C01810=1180.167,97.495,-51.204,-178.948,6.146,148.795
C01811=1180.172,97.245,-51.186,-178.951,6.145,148.796
C01812=1180.177,96.996,-51.166,-178.954,6.143,148.797
C01813=1180.182,96.747,-51.148,-178.957,6.142,148.797
C01814=1180.187,96.498,-51.130,-178.959,6.141,148.798
C01815=1180.192,96.249,-51.112,-178.962,6.139,148.798
C01816=1180.197,95.999,-51.094,-178.964,6.139,148.799
C01817=1180.201,95.750,-51.076,-178.967,6.137,148.799
C01818=1180.206,95.500,-51.058,-178.970,6.136,148.800
C01819=1180.211,95.251,-51.040,-178.973,6.135,148.800
C01820=1180.217,95.002,-51.021,-178.975,6.134,148.801
C01821=1180.221,94.753,-51.003,-178.978,6.132,148.801
C01822=1180.226,94.503,-50.985,-178.980,6.132,148.802
C01823=1180.231,94.254,-50.967,-178.983,6.130,148.802
C01824=1180.236,94.004,-50.949,-178.985,6.129,148.803
C01825=1180.240,93.755,-50.931,-178.989,6.128,148.803
C01826=1180.245,93.506,-50.913,-178.991,6.127,148.804
C01827=1180.250,93.257,-50.895,-178.993,6.125,148.804
C01828=1180.255,93.008,-50.877,-178.996,6.125,148.805
C01829=1180.260,92.758,-50.859,-178.999,6.123,148.805
C01830=1180.264,92.509,-50.841,-179.002,6.122,148.806
C01831=1180.269,92.259,-50.823,-179.004,6.121,148.806
C01832=1180.274,92.010,-50.805,-179.007,6.119,148.807
C01833=1180.279,91.761,-50.787,-179.009,6.118,148.807
C01834=1180.284,91.512,-50.769,-179.012,6.117,148.808
C01835=1180.289,91.263,-50.751,-179.015,6.116,148.808
C01836=1180.294,91.013,-50.734,-179.017,6.114,148.809
C01837=1180.299,90.764,-50.716,-179.020,6.114,148.809
C01838=1180.304,90.515,-50.698,-179.023,6.112,148.810
C01839=1180.309,90.265,-50.680,-179.025,6.112,148.811
C01840=1180.313,90.016,-50.661,-179.028,6.110,148.811
C01841=1180.318,89.766,-50.643,-179.030,6.109,148.811
C01842=1180.323,89.517,-50.625,-179.034,6.108,148.812
C01843=1180.328,89.267,-50.608,-179.036,6.107,148.812
C01844=1180.333,89.018,-50.590,-179.039,6.105,148.813
C01845=1180.338,88.769,-50.572,-179.041,6.105,148.814
C01846=1180.342,88.520,-50.555,-179.044,6.103,148.814
C01847=1180.347,88.271,-50.537,-179.046,6.102,148.815
C01848=1180.352,88.021,-50.520,-179.050,6.101,148.815
C01849=1180.357,87.772,-50.502,-179.052,6.100,148.816
C01850=1180.362,87.523,-50.484,-179.054,6.099,148.816
C01851=1180.367,87.274,-50.466,-179.057,6.098,148.817
C01852=1180.372,87.024,-50.448,-179.059,6.097,148.817
C01853=1180.377,86.775,-50.430,-179.062,6.096,148.818
C01854=1180.382,86.526,-50.412,-179.064,6.095,148.818
C01855=1180.387,86.276,-50.396,-179.068,6.093,148.819
C01856=1180.392,86.027,-50.378,-179.070,6.092,148.819
C01857=1180.397,85.778,-50.360,-179.073,6.091,148.820
C01858=1180.402,85.528,-50.343,-179.075,6.090,148.820
C01859=1180.407,85.279,-50.325,-179.078,6.089,148.821
C01860=1180.412,85.030,-50.307,-179.081,6.088,148.821
C01861=1180.416,84.780,-50.290,-179.083,6.086,148.822
C01862=1180.421,84.531,-50.272,-179.086,6.086,148.823
C01863=1180.426,84.282,-50.254,-179.089,6.084,148.823
C01864=1180.431,84.032,-50.237,-179.091,6.083,148.824
C01865=1180.436,83.783,-50.219,-179.094,6.082,148.824
C01866=1180.440,83.533,-50.202,-179.097,6.081,148.825
C01867=1180.445,83.284,-50.184,-179.099,6.080,148.825
C01868=1180.450,83.035,-50.166,-179.102,6.079,148.826
C01869=1180.456,82.785,-50.149,-179.104,6.078,148.826
C01870=1180.460,82.536,-50.131,-179.107,6.077,148.827
C01871=1180.465,82.286,-50.114,-179.109,6.076,148.827
C01872=1180.470,82.037,-50.096,-179.113,6.074,148.828
C01873=1180.475,81.787,-50.079,-179.115,6.073,148.828
C01874=1180.479,81.539,-50.062,-179.118,6.072,148.829
C01875=1180.484,81.289,-50.044,-179.120,6.071,148.829
C01876=1180.489,81.040,-50.026,-179.123,6.071,148.830
C01877=1180.495,80.771,-50.008,-179.125,6.069,148.830
C01878=1180.500,80.504,-49.989,-179.129,6.068,148.831
C01879=1180.505,80.235,-49.970,-179.131,6.067,148.832
C01880=1180.511,79.966,-49.952,-179.134,6.065,148.832
C01881=1180.516,79.717,-49.934,-179.137,6.065,148.833
C01882=1180.520,79.468,-49.918,-179.139,6.063,148.833
C01883=1180.525,79.219,-49.900,-179.142,6.063,148.834
C01884=1180.531,78.969,-49.882,-179.145,6.061,148.834
C01885=1180.535,78.719,-49.866,-179.147,6.060,148.835
C01886=1180.540,78.470,-49.848,-179.150,6.059,148.835
C01887=1180.545,78.220,-49.830,-179.153,6.058,148.836
C01888=1180.550,77.972,-49.813,-179.155,6.057,148.837
C01889=1180.555,77.722,-49.796,-179.158,6.056,148.837
C01890=1180.560,77.473,-49.779,-179.160,6.055,148.838
C01891=1180.565,77.224,-49.761,-179.163,6.054,148.838
C01892=1180.570,76.974,-49.744,-179.166,6.053,148.839
C01893=1180.574,76.724,-49.727,-179.168,6.052,148.839
C01894=1180.579,76.475,-49.710,-179.171,6.050,148.840
C01895=1180.584,76.227,-49.693,-179.174,6.050,148.840
C01896=1180.589,75.977,-49.676,-179.176,6.048,148.841
C01897=1180.594,75.728,-49.658,-179.179,6.048,148.841
C01898=1180.599,75.478,-49.641,-179.182,6.046,148.842
C01899=1180.604,75.228,-49.624,-179.184,6.045,148.843
C01900=1180.609,74.979,-49.607,-179.186,6.045,148.843
C01901=1180.614,74.730,-49.590,-179.190,6.043,148.844
C01902=1180.619,74.481,-49.573,-179.192,6.042,148.844
C01903=1180.624,74.231,-49.556,-179.195,6.041,148.845
C01904=1180.628,73.982,-49.539,-179.197,6.040,148.845
C01905=1180.633,73.732,-49.521,-179.200,6.040,148.846
C01906=1180.639,73.483,-49.504,-179.202,6.038,148.846
C01907=1180.643,73.234,-49.488,-179.205,6.037,148.847
C01908=1180.649,72.984,-49.470,-179.207,6.036,148.847
C01909=1180.653,72.735,-49.454,-179.210,6.035,148.848
C01910=1180.658,72.485,-49.436,-179.213,6.034,148.848
C01911=1180.663,72.237,-49.419,-179.216,6.033,148.849
C01912=1180.668,71.987,-49.403,-179.218,6.032,148.850
C01913=1180.673,71.737,-49.385,-179.221,6.031,148.850
C01914=1180.677,71.488,-49.369,-179.223,6.030,148.851
C01915=1180.683,71.239,-49.352,-179.226,6.029,148.851
C01916=1180.688,70.989,-49.335,-179.229,6.027,148.852
C01917=1180.693,70.739,-49.318,-179.231,6.027,148.852
C01918=1180.697,70.491,-49.301,-179.233,6.026,148.853
C01919=1180.703,70.241,-49.284,-179.237,6.025,148.853
C01920=1180.707,69.992,-49.267,-179.239,6.024,148.854
C01921=1180.712,69.743,-49.250,-179.241,6.023,148.855
C01922=1180.718,69.493,-49.233,-179.244,6.022,148.855
C01923=1180.722,69.244,-49.217,-179.247,6.021,148.856
C01924=1180.727,68.994,-49.199,-179.250,6.020,148.856
C01925=1180.732,68.745,-49.183,-179.252,6.019,148.857
C01926=1180.737,68.496,-49.167,-179.255,6.018,148.857
C01927=1180.742,68.246,-49.149,-179.257,6.017,148.858
C01928=1180.747,67.997,-49.133,-179.260,6.016,148.858
C01929=1180.752,67.748,-49.116,-179.262,6.015,148.859
C01930=1180.757,67.498,-49.099,-179.265,6.014,148.860
C01931=1180.761,67.249,-49.082,-179.268,6.013,148.860
C01932=1180.767,66.999,-49.065,-179.270,6.012,148.861
C01933=1180.772,66.750,-49.049,-179.273,6.011,148.861
C01934=1180.776,66.500,-49.032,-179.276,6.010,148.862
C01935=1180.781,66.251,-49.015,-179.278,6.009,148.862
C01936=1180.786,66.002,-48.999,-179.281,6.008,148.863
C01937=1180.791,65.752,-48.982,-179.283,6.007,148.863
C01938=1180.796,65.503,-48.965,-179.286,6.007,148.864
C01939=1180.802,65.253,-48.949,-179.289,6.005,148.865
C01940=1180.806,65.004,-48.932,-179.291,6.004,148.865
C01941=1180.810,64.754,-48.916,-179.294,6.003,148.866
C01942=1180.816,64.505,-48.899,-179.296,6.002,148.866
C01943=1180.821,64.256,-48.882,-179.299,6.002,148.867
C01944=1180.826,64.007,-48.866,-179.302,6.000,148.867
C01945=1180.830,63.757,-48.849,-179.304,5.999,148.868
C01946=1180.836,63.507,-48.833,-179.307,5.998,148.868
C01947=1180.841,63.258,-48.816,-179.310,5.997,148.869
C01948=1180.845,63.009,-48.800,-179.312,5.997,148.870
C01949=1180.850,62.759,-48.783,-179.315,5.996,148.870
C01950=1180.856,62.510,-48.766,-179.318,5.994,148.871
C01951=1180.860,62.261,-48.749,-179.320,5.993,148.871
C01952=1180.866,62.011,-48.734,-179.323,5.993,148.872
C01953=1180.870,61.762,-48.717,-179.325,5.992,148.872
C01954=1180.875,61.512,-48.700,-179.328,5.991,148.873
C01955=1180.880,61.263,-48.684,-179.330,5.990,148.873
C01956=1180.885,61.013,-48.668,-179.333,5.989,148.874
C01957=1180.890,60.764,-48.651,-179.336,5.988,148.875
C01958=1180.895,60.515,-48.635,-179.338,5.987,148.875
C01959=1180.900,60.266,-48.618,-179.341,5.987,148.876
C01960=1180.905,60.016,-48.602,-179.343,5.985,148.876
C01961=1180.910,59.766,-48.585,-179.346,5.984,148.877
C01962=1180.915,59.517,-48.569,-179.348,5.984,148.877
C01963=1180.920,59.267,-48.553,-179.351,5.982,148.878
C01964=1180.925,59.018,-48.537,-179.354,5.981,148.878
C01965=1180.929,58.769,-48.520,-179.356,5.981,148.879
C01966=1180.935,58.520,-48.504,-179.359,5.979,148.880
C01967=1180.940,58.270,-48.487,-179.362,5.979,148.880
C01968=1180.945,58.021,-48.471,-179.364,5.978,148.881
C01969=1180.950,57.771,-48.455,-179.366,5.977,148.881
C01970=1180.955,57.522,-48.438,-179.370,5.976,148.882
C01971=1180.960,57.272,-48.423,-179.372,5.975,148.882
C01972=1180.965,57.023,-48.406,-179.374,5.974,148.883
C01973=1180.969,56.774,-48.390,-179.378,5.973,148.884
C01974=1180.975,56.524,-48.374,-179.380,5.972,148.884
C01975=1180.979,56.275,-48.357,-179.382,5.972,148.885
C01976=1180.984,56.025,-48.342,-179.385,5.971,148.885
C01977=1180.990,55.776,-48.324,-179.388,5.969,148.886
C01978=1180.995,55.526,-48.309,-179.390,5.969,148.886
C01979=1180.999,55.277,-48.292,-179.393,5.968,148.887
C01980=1181.005,55.027,-48.277,-179.396,5.967,148.888
C01981=1181.010,54.759,-48.258,-179.398,5.966,148.888
C01982=1181.015,54.490,-48.241,-179.401,5.965,148.889
C01983=1181.021,54.222,-48.224,-179.404,5.964,148.889
C01984=1181.026,53.953,-48.207,-179.406,5.964,148.890
C01985=1181.031,53.704,-48.191,-179.409,5.962,148.891
C01986=1181.036,53.454,-48.175,-179.412,5.961,148.891
C01987=1181.041,53.205,-48.159,-179.414,5.961,148.892
C01988=1181.046,52.956,-48.143,-179.417,5.960,148.892
C01989=1181.050,52.706,-48.126,-179.420,5.959,148.893
C01990=1181.056,52.457,-48.111,-179.422,5.958,148.893
C01991=1181.060,52.207,-48.094,-179.425,5.957,148.894
C01992=1181.066,51.958,-48.078,-179.427,5.956,148.895
C01993=1181.071,51.708,-48.063,-179.430,5.955,148.895
C01994=1181.076,51.459,-48.046,-179.433,5.954,148.896
C01995=1181.081,51.210,-48.031,-179.435,5.954,148.896
C01996=1181.085,50.960,-48.014,-179.438,5.952,148.897
C01997=1181.091,50.711,-47.998,-179.440,5.951,148.897
C01998=1181.095,50.461,-47.983,-179.443,5.951,148.898
C01999=1181.100,50.212,-47.967,-179.445,5.950,148.899
C02000=1181.105,49.963,-47.951,-179.448,5.949,148.899
C02001=1181.110,49.713,-47.935,-179.451,5.948,148.900
C02002=1181.115,49.464,-47.919,-179.453,5.947,148.900
C02003=1181.120,49.214,-47.903,-179.456,5.947,148.901
C02004=1181.125,48.964,-47.887,-179.459,5.945,148.902
C02005=1181.130,48.716,-47.871,-179.461,5.945,148.902
C02006=1181.135,48.465,-47.855,-179.464,5.944,148.903
C02007=1181.140,48.216,-47.840,-179.466,5.943,148.903
C02008=1181.145,47.967,-47.824,-179.469,5.942,148.904
C02009=1181.150,47.717,-47.808,-179.472,5.941,148.905
C02010=1181.155,47.468,-47.792,-179.474,5.940,148.905
C02011=1181.160,47.219,-47.777,-179.476,5.940,148.906
C02012=1181.165,46.969,-47.761,-179.479,5.939,148.906
C02013=1181.170,46.720,-47.745,-179.482,5.938,148.907
C02014=1181.175,46.471,-47.729,-179.484,5.937,148.907
C02015=1181.180,46.221,-47.713,-179.487,5.936,148.908
C02016=1181.185,45.971,-47.698,-179.489,5.936,148.909
C02017=1181.191,45.722,-47.682,-179.492,5.934,148.909
C02018=1181.194,45.473,-47.666,-179.495,5.934,148.910
C02019=1181.200,45.223,-47.651,-179.497,5.933,148.910
C02020=1181.205,44.974,-47.635,-179.499,5.932,148.911
C02021=1181.210,44.724,-47.619,-179.503,5.931,148.911
C02022=1181.215,44.474,-47.603,-179.505,5.930,148.912
C02023=1181.220,44.225,-47.588,-179.507,5.930,148.913
C02024=1181.225,43.975,-47.572,-179.510,5.929,148.913
C02025=1181.230,43.726,-47.556,-179.512,5.928,148.914
C02026=1181.235,43.477,-47.541,-179.515,5.927,148.914
C02027=1181.239,43.227,-47.525,-179.518,5.926,148.915
C02028=1181.245,42.978,-47.510,-179.520,5.926,148.915
C02029=1181.250,42.728,-47.494,-179.523,5.925,148.916
C02030=1181.255,42.479,-47.478,-179.525,5.924,148.917
C02031=1181.259,42.229,-47.463,-179.528,5.923,148.917
C02032=1181.265,41.980,-47.447,-179.531,5.922,148.918
C02033=1181.270,41.730,-47.432,-179.533,5.921,148.918
C02034=1181.275,41.481,-47.417,-179.536,5.921,148.919
C02035=1181.280,41.231,-47.401,-179.538,5.920,148.920
C02036=1181.285,40.982,-47.385,-179.541,5.919,148.920
C02037=1181.290,40.733,-47.370,-179.544,5.918,148.921
C02038=1181.295,40.483,-47.355,-179.546,5.917,148.921
C02039=1181.300,40.233,-47.339,-179.548,5.917,148.922
C02040=1181.304,39.984,-47.324,-179.551,5.916,148.923
C02041=1181.310,39.735,-47.308,-179.554,5.915,148.923
C02042=1181.315,39.485,-47.293,-179.557,5.914,148.924
C02043=1181.320,39.236,-47.278,-179.559,5.914,148.924
C02044=1181.325,38.986,-47.262,-179.561,5.913,148.925
C02045=1181.330,38.737,-47.246,-179.564,5.912,148.926
C02046=1181.335,38.487,-47.231,-179.567,5.911,148.926
C02047=1181.340,38.238,-47.216,-179.569,5.910,148.927
C02048=1181.346,37.989,-47.200,-179.572,5.910,148.927
C02049=1181.350,37.739,-47.185,-179.574,5.909,148.928
C02050=1181.355,37.489,-47.170,-179.577,5.908,148.928
C02051=1181.360,37.240,-47.155,-179.579,5.908,148.929
C02052=1181.365,36.990,-47.139,-179.582,5.906,148.930
C02053=1181.371,36.741,-47.124,-179.585,5.906,148.930
C02054=1181.375,36.491,-47.108,-179.587,5.905,148.931
C02055=1181.380,36.242,-47.093,-179.590,5.904,148.931
C02056=1181.385,35.993,-47.078,-179.592,5.904,148.932
C02057=1181.390,35.743,-47.063,-179.594,5.903,148.932
C02058=1181.395,35.494,-47.048,-179.598,5.902,148.933
C02059=1181.400,35.244,-47.032,-179.600,5.901,148.934
C02060=1181.405,34.994,-47.017,-179.602,5.900,148.934
C02061=1181.410,34.745,-47.001,-179.605,5.900,148.935
C02062=1181.416,34.495,-46.986,-179.608,5.899,148.936
C02063=1181.420,34.246,-46.971,-179.610,5.898,148.936
C02064=1181.426,33.996,-46.956,-179.613,5.897,148.937
C02065=1181.430,33.747,-46.941,-179.616,5.896,148.937
C02066=1181.436,33.497,-46.926,-179.618,5.896,148.938
C02067=1181.441,33.248,-46.911,-179.621,5.895,148.939
C02068=1181.445,32.998,-46.895,-179.623,5.895,148.939
C02069=1181.450,32.749,-46.880,-179.625,5.894,148.940
C02070=1181.456,32.499,-46.865,-179.629,5.892,148.940
C02071=1181.460,32.250,-46.850,-179.631,5.892,148.941
C02072=1181.465,32.001,-46.835,-179.633,5.891,148.941
C02073=1181.471,31.751,-46.820,-179.636,5.891,148.942
C02074=1181.475,31.502,-46.805,-179.638,5.890,148.943
C02075=1181.481,31.252,-46.790,-179.641,5.889,148.943
C02076=1181.485,31.003,-46.775,-179.643,5.889,148.944
C02077=1181.491,30.753,-46.760,-179.646,5.887,148.944
C02078=1181.495,30.503,-46.744,-179.649,5.887,148.945
C02079=1181.500,30.254,-46.730,-179.652,5.886,148.946
C02080=1181.506,30.004,-46.715,-179.654,5.885,148.946
C02081=1181.510,29.755,-46.700,-179.656,5.885,148.947
C02082=1181.516,29.505,-46.685,-179.659,5.884,148.948
C02083=1181.521,29.256,-46.670,-179.661,5.883,148.948
C02084=1181.526,29.007,-46.654,-179.664,5.882,148.949
C02085=1181.531,28.738,-46.638,-179.667,5.882,148.949
C02086=1181.536,28.469,-46.623,-179.670,5.881,148.950
C02087=1181.542,28.200,-46.606,-179.672,5.880,148.951
C02088=1181.547,27.931,-46.591,-179.675,5.879,148.951
C02089=1181.553,27.682,-46.575,-179.678,5.878,148.952
C02090=1181.557,27.432,-46.561,-179.680,5.878,148.953
C02091=1181.562,27.183,-46.546,-179.682,5.877,148.953
C02092=1181.568,26.933,-46.531,-179.685,5.877,148.954
C02093=1181.572,26.684,-46.516,-179.688,5.876,148.954
C02094=1181.577,26.434,-46.502,-179.690,5.875,148.955
C02095=1181.583,26.185,-46.486,-179.693,5.874,148.955
C02096=1181.588,25.935,-46.472,-179.696,5.873,148.956
C02097=1181.592,25.686,-46.457,-179.698,5.873,148.957
C02098=1181.598,25.436,-46.442,-179.701,5.872,148.957
C02099=1181.603,25.187,-46.427,-179.703,5.872,148.958
C02100=1181.608,24.937,-46.413,-179.705,5.871,148.958
C02101=1181.612,24.688,-46.398,-179.708,5.870,148.959
C02102=1181.618,24.438,-46.383,-179.711,5.870,148.960
C02103=1181.623,24.188,-46.369,-179.713,5.869,148.960
C02104=1181.628,23.939,-46.354,-179.716,5.868,148.961
C02105=1181.633,23.689,-46.339,-179.719,5.867,148.962
C02106=1181.638,23.440,-46.324,-179.721,5.866,148.962
C02107=1181.643,23.190,-46.309,-179.724,5.866,148.963
C02108=1181.648,22.941,-46.295,-179.726,5.865,148.963
C02109=1181.653,22.691,-46.280,-179.728,5.864,148.964
C02110=1181.658,22.442,-46.265,-179.731,5.864,148.965
C02111=1181.663,22.193,-46.250,-179.734,5.863,148.965
C02112=1181.668,21.943,-46.236,-179.736,5.863,148.966
C02113=1181.673,21.694,-46.222,-179.738,5.862,148.966
C02114=1181.679,21.444,-46.207,-179.741,5.862,148.967
C02115=1181.684,21.195,-46.192,-179.743,5.861,148.967
C02116=1181.689,20.945,-46.178,-179.747,5.859,148.968
C02117=1181.693,20.696,-46.163,-179.749,5.859,148.969
C02118=1181.698,20.446,-46.149,-179.751,5.858,148.969
C02119=1181.704,20.196,-46.134,-179.754,5.858,148.970
C02120=1181.709,19.946,-46.120,-179.757,5.857,148.971
C02121=1181.714,19.697,-46.105,-179.759,5.856,148.971
C02122=1181.719,19.448,-46.090,-179.761,5.856,148.972
C02123=1181.724,19.198,-46.076,-179.764,5.855,148.972
C02124=1181.729,18.949,-46.062,-179.766,5.854,148.973
C02125=1181.734,18.700,-46.046,-179.769,5.854,148.974
C02126=1181.739,18.450,-46.032,-179.772,5.853,148.974
C02127=1181.744,18.200,-46.018,-179.774,5.853,148.975
C02128=1181.749,17.950,-46.004,-179.777,5.851,148.975
C02129=1181.754,17.701,-45.989,-179.780,5.851,148.976
C02130=1181.759,17.452,-45.974,-179.782,5.850,148.977
C02131=1181.764,17.202,-45.960,-179.784,5.849,148.977
C02132=1181.769,16.952,-45.946,-179.787,5.849,148.978
C02133=1181.774,16.703,-45.932,-179.789,5.848,148.978
C02134=1181.779,16.453,-45.918,-179.792,5.848,148.979
C02135=1181.785,16.204,-45.902,-179.795,5.847,148.980
C02136=1181.790,15.954,-45.888,-179.797,5.846,148.980
C02137=1181.795,15.705,-45.874,-179.799,5.846,148.981
C02138=1181.800,15.455,-45.859,-179.802,5.845,148.982
C02139=1181.805,15.206,-45.845,-179.805,5.845,148.982
C02140=1181.810,14.956,-45.831,-179.807,5.844,148.983
C02141=1181.815,14.706,-45.817,-179.809,5.843,148.983
C02142=1181.820,14.457,-45.802,-179.812,5.843,148.984
C02143=1181.825,14.208,-45.787,-179.814,5.842,148.985
C02144=1181.830,13.958,-45.773,-179.817,5.842,148.985
C02145=1181.835,13.709,-45.759,-179.820,5.841,148.986
C02146=1181.840,13.459,-45.745,-179.822,5.839,148.986
C02147=1181.845,13.210,-45.731,-179.825,5.839,148.987
C02148=1181.850,12.960,-45.716,-179.828,5.839,148.988
C02149=1181.855,12.710,-45.702,-179.830,5.838,148.988
C02150=1181.861,12.461,-45.688,-179.832,5.837,148.989
C02151=1181.866,12.211,-45.674,-179.835,5.837,148.990
C02152=1181.870,11.962,-45.660,-179.837,5.836,148.990
C02153=1181.875,11.712,-45.645,-179.840,5.835,148.991
C02154=1181.881,11.463,-45.632,-179.843,5.835,148.991
C02155=1181.886,11.213,-45.617,-179.845,5.834,148.992
C02156=1181.891,10.964,-45.603,-179.847,5.834,148.993
C02157=1181.896,10.714,-45.589,-179.850,5.833,148.993
C02158=1181.901,10.464,-45.574,-179.853,5.833,148.994
C02159=1181.906,10.215,-45.561,-179.855,5.832,148.994
C02160=1181.911,9.965,-45.546,-179.858,5.831,148.995
C02161=1181.916,9.716,-45.532,-179.860,5.831,148.996
C02162=1181.921,9.466,-45.518,-179.862,5.830,148.996
C02163=1181.926,9.217,-45.505,-179.865,5.829,148.997
C02164=1181.931,8.967,-45.491,-179.868,5.829,148.998
C02165=1181.936,8.717,-45.477,-179.870,5.828,148.998
C02166=1181.942,8.468,-45.463,-179.872,5.828,148.999
C02167=1181.947,8.219,-45.448,-179.875,5.827,148.999
C02168=1181.952,7.969,-45.434,-179.877,5.826,149.000
C02169=1181.957,7.719,-45.420,-179.880,5.826,149.001
C02170=1181.962,7.470,-45.406,-179.883,5.825,149.001
C02171=1181.967,7.220,-45.392,-179.885,5.825,149.002
C02172=1181.972,6.970,-45.379,-179.887,5.824,149.002
C02173=1181.977,6.721,-45.365,-179.890,5.824,149.003
C02174=1181.982,6.472,-45.350,-179.893,5.823,149.004
C02175=1181.987,6.222,-45.336,-179.895,5.822,149.004
C02176=1181.992,5.972,-45.322,-179.898,5.822,149.005
C02177=1181.998,5.723,-45.309,-179.900,5.821,149.006
C02178=1182.002,5.473,-45.295,-179.902,5.820,149.006
C02179=1182.007,5.223,-45.281,-179.905,5.820,149.007
C02180=1182.013,4.974,-45.267,-179.908,5.819,149.007
C02181=1182.018,4.725,-45.253,-179.910,5.819,149.008
C02182=1182.023,4.474,-45.239,-179.912,5.818,149.009
C02183=1182.028,4.226,-45.226,-179.915,5.818,149.009
C02184=1182.033,3.976,-45.211,-179.918,5.817,149.010
C02185=1182.038,3.726,-45.197,-179.920,5.816,149.010
C02186=1182.044,3.477,-45.184,-179.923,5.816,149.011
C02187=1182.048,3.227,-45.170,-179.925,5.815,149.012
C02188=1182.053,2.978,-45.156,-179.927,5.815,149.012
C02189=1182.059,2.709,-45.141,-179.930,5.814,149.013
C02190=1182.064,2.439,-45.126,-179.933,5.814,149.014
C02191=1182.070,2.170,-45.111,-179.936,5.812,149.014
C02192=1182.075,1.901,-45.096,-179.939,5.812,149.015
C02193=1182.081,1.651,-45.083,-179.941,5.811,149.016
C02194=1182.085,1.402,-45.069,-179.943,5.811,149.016
C02195=1182.091,1.153,-45.056,-179.946,5.810,149.017
C02196=1182.096,0.902,-45.042,-179.949,5.810,149.017
C02197=1182.101,0.653,-45.028,-179.951,5.809,149.018
C02198=1182.106,0.404,-45.014,-179.954,5.808,149.019
C02199=1182.111,0.154,-45.001,-179.956,5.808,149.019
C02200=1182.117,-0.095,-44.987,-179.959,5.807,149.020
C02201=1182.121,-0.345,-44.973,-179.961,5.806,149.020
C02202=1182.126,-0.595,-44.960,-179.964,5.806,149.021
C02203=1182.132,-0.844,-44.946,-179.966,5.806,149.022
C02204=1182.136,-1.094,-44.933,-179.968,5.805,149.022
C02205=1182.142,-1.343,-44.919,-179.971,5.805,149.023
C02206=1182.147,-1.594,-44.905,-179.973,5.805,149.024
C02207=1182.151,-1.843,-44.892,-179.976,5.804,149.024
C02208=1182.157,-2.092,-44.878,-179.978,5.803,149.025
C02209=1182.162,-2.342,-44.864,-179.981,5.803,149.026
C02210=1182.167,-2.591,-44.851,-179.983,5.802,149.026
C02211=1182.172,-2.841,-44.837,-179.986,5.801,149.027
C02212=1182.178,-3.090,-44.823,-179.988,5.801,149.027
C02213=1182.182,-3.340,-44.810,-179.991,5.801,149.028
C02214=1182.188,-3.589,-44.797,-179.993,5.800,149.029
C02215=1182.192,-3.839,-44.784,-179.996,5.799,149.029
C02216=1182.198,-4.088,-44.770,-179.998,5.799,149.030
C02217=1182.203,-4.339,-44.756,179.999,5.798,149.031
C02218=1182.207,-4.588,-44.742,179.997,5.797,149.031
C02219=1182.213,-4.838,-44.729,179.994,5.797,149.032
C02220=1182.218,-5.088,-44.716,179.992,5.796,149.032
C02221=1182.223,-5.337,-44.702,179.989,5.796,149.033
C02222=1182.228,-5.587,-44.689,179.987,5.795,149.034
C02223=1182.233,-5.836,-44.675,179.984,5.795,149.034
C02224=1182.238,-6.086,-44.662,179.981,5.794,149.035
C02225=1182.243,-6.335,-44.649,179.979,5.793,149.035
C02226=1182.249,-6.585,-44.635,179.977,5.794,149.036
C02227=1182.254,-6.834,-44.622,179.975,5.793,149.037
C02228=1182.259,-7.084,-44.608,179.972,5.792,149.037
C02229=1182.264,-7.334,-44.596,179.970,5.792,149.038
C02230=1182.269,-7.584,-44.582,179.967,5.792,149.039
C02231=1182.274,-7.833,-44.569,179.965,5.791,149.039
C02232=1182.280,-8.082,-44.555,179.962,5.790,149.040
C02233=1182.284,-8.332,-44.543,179.960,5.790,149.041
C02234=1182.290,-8.581,-44.529,179.957,5.789,149.041
C02235=1182.294,-8.831,-44.516,179.955,5.788,149.042
C02236=1182.300,-9.081,-44.502,179.952,5.788,149.042
C02237=1182.304,-9.330,-44.489,179.949,5.788,149.043
C02238=1182.310,-9.580,-44.476,179.947,5.787,149.044
C02239=1182.315,-9.830,-44.463,179.945,5.786,149.044
C02240=1182.320,-10.079,-44.449,179.942,5.786,149.045
C02241=1182.325,-10.329,-44.436,179.940,5.786,149.046
C02242=1182.331,-10.579,-44.423,179.938,5.785,149.046
C02243=1182.336,-10.828,-44.410,179.935,5.785,149.047
C02244=1182.341,-11.078,-44.396,179.932,5.784,149.047
C02245=1182.346,-11.327,-44.383,179.930,5.783,149.048
C02246=1182.350,-11.577,-44.370,179.928,5.783,149.049
C02247=1182.356,-11.827,-44.357,179.925,5.783,149.049
C02248=1182.360,-12.076,-44.343,179.922,5.782,149.050
C02249=1182.366,-12.326,-44.330,179.920,5.781,149.050
C02250=1182.371,-12.575,-44.317,179.917,5.781,149.051
C02251=1182.377,-12.825,-44.304,179.915,5.780,149.052
C02252=1182.382,-13.075,-44.291,179.913,5.779,149.052
C02253=1182.386,-13.324,-44.278,179.910,5.780,149.053
C02254=1182.392,-13.574,-44.264,179.908,5.779,149.054
C02255=1182.397,-13.823,-44.252,179.905,5.779,149.054
C02256=1182.402,-14.073,-44.239,179.903,5.778,149.055
C02257=1182.407,-14.323,-44.226,179.900,5.778,149.056
C02258=1182.412,-14.573,-44.213,179.898,5.777,149.056
C02259=1182.418,-14.822,-44.199,179.895,5.776,149.057
C02260=1182.423,-15.071,-44.186,179.893,5.776,149.057
C02261=1182.427,-15.321,-44.173,179.890,5.775,149.058
C02262=1182.433,-15.571,-44.160,179.888,5.775,149.059
C02263=1182.438,-15.820,-44.147,179.886,5.775,149.059
C02264=1182.443,-16.070,-44.134,179.883,5.774,149.060
C02265=1182.449,-16.319,-44.121,179.881,5.774,149.061
C02266=1182.454,-16.569,-44.109,179.878,5.773,149.061
C02267=1182.458,-16.819,-44.096,179.876,5.773,149.062
C02268=1182.464,-17.068,-44.082,179.873,5.772,149.062
C02269=1182.469,-17.318,-44.070,179.870,5.772,149.063
C02270=1182.473,-17.567,-44.056,179.868,5.771,149.064
C02271=1182.479,-17.816,-44.044,179.866,5.770,149.064
C02272=1182.484,-18.066,-44.030,179.864,5.771,149.065
C02273=1182.489,-18.316,-44.017,179.861,5.770,149.065
C02274=1182.494,-18.565,-44.005,179.859,5.770,149.066
C02275=1182.500,-18.815,-43.992,179.856,5.769,149.067
C02276=1182.504,-19.065,-43.979,179.854,5.768,149.067
C02277=1182.510,-19.314,-43.966,179.851,5.768,149.068
C02278=1182.515,-19.564,-43.953,179.849,5.767,149.069
C02279=1182.521,-19.813,-43.940,179.846,5.767,149.069
C02280=1182.525,-20.063,-43.927,179.844,5.767,149.070
C02281=1182.530,-20.313,-43.915,179.842,5.766,149.071
C02282=1182.536,-20.563,-43.903,179.839,5.766,149.071
C02283=1182.541,-20.813,-43.889,179.837,5.765,149.072
C02284=1182.546,-21.062,-43.877,179.834,5.765,149.072
C02285=1182.551,-21.312,-43.864,179.832,5.764,149.073
C02286=1182.556,-21.561,-43.851,179.829,5.764,149.074
C02287=1182.561,-21.811,-43.838,179.827,5.763,149.074
C02288=1182.567,-22.061,-43.825,179.825,5.763,149.075
C02289=1182.572,-22.310,-43.813,179.822,5.763,149.076
C02290=1182.577,-22.559,-43.800,179.820,5.762,149.076
C02291=1182.581,-22.809,-43.787,179.817,5.762,149.077
C02292=1182.586,-23.059,-43.774,179.814,5.761,149.078
C02293=1182.593,-23.329,-43.761,179.812,5.761,149.078
C02294=1182.598,-23.598,-43.748,179.809,5.760,149.079
C02295=1182.604,-23.868,-43.733,179.806,5.760,149.080
C02296=1182.609,-24.138,-43.720,179.804,5.759,149.080
C02297=1182.614,-24.387,-43.707,179.802,5.758,149.081
C02298=1182.619,-24.637,-43.694,179.799,5.758,149.082
C02299=1182.625,-24.887,-43.683,179.797,5.758,149.082
C02300=1182.630,-25.136,-43.669,179.795,5.758,149.083
C02301=1182.635,-25.386,-43.656,179.792,5.757,149.083
C02302=1182.640,-25.636,-43.644,179.789,5.757,149.084
C02303=1182.645,-25.885,-43.631,179.787,5.756,149.085
C02304=1182.651,-26.135,-43.619,179.785,5.755,149.085
C02305=1182.655,-26.385,-43.606,179.782,5.755,149.086
C02306=1182.660,-26.634,-43.594,179.780,5.755,149.087
C02307=1182.665,-26.883,-43.581,179.778,5.754,149.087
C02308=1182.671,-27.133,-43.569,179.775,5.754,149.088
C02309=1182.676,-27.383,-43.557,179.772,5.754,149.088
C02310=1182.681,-27.632,-43.544,179.770,5.753,149.089
C02311=1182.686,-27.882,-43.530,179.767,5.752,149.090
C02312=1182.692,-28.132,-43.519,179.765,5.753,149.090
C02313=1182.697,-28.382,-43.506,179.763,5.752,149.091
C02314=1182.702,-28.631,-43.493,179.761,5.751,149.092
C02315=1182.707,-28.881,-43.482,179.758,5.751,149.092
C02316=1182.712,-29.131,-43.469,179.755,5.750,149.093
C02317=1182.717,-29.380,-43.456,179.753,5.750,149.094
C02318=1182.723,-29.630,-43.444,179.751,5.750,149.094
C02319=1182.728,-29.879,-43.431,179.748,5.749,149.095
C02320=1182.733,-30.129,-43.419,179.746,5.749,149.095
C02321=1182.738,-30.379,-43.407,179.744,5.748,149.096
C02322=1182.743,-30.628,-43.394,179.741,5.748,149.097
C02323=1182.748,-30.878,-43.381,179.738,5.747,149.097
C02324=1182.753,-31.128,-43.370,179.736,5.748,149.098
C02325=1182.758,-31.377,-43.357,179.734,5.747,149.099
C02326=1182.764,-31.627,-43.344,179.731,5.746,149.099
C02327=1182.769,-31.877,-43.332,179.729,5.746,149.100
C02328=1182.774,-32.126,-43.320,179.726,5.745,149.100
C02329=1182.780,-32.376,-43.308,179.724,5.745,149.101
C02330=1182.785,-32.625,-43.295,179.722,5.745,149.102
C02331=1182.790,-32.875,-43.283,179.719,5.745,149.102
C02332=1182.795,-33.125,-43.270,179.717,5.744,149.103
C02333=1182.800,-33.374,-43.258,179.714,5.743,149.104
C02334=1182.805,-33.624,-43.246,179.712,5.743,149.104
C02335=1182.810,-33.873,-43.234,179.710,5.743,149.105
C02336=1182.815,-34.123,-43.222,179.707,5.742,149.106
C02337=1182.820,-34.373,-43.210,179.705,5.742,149.106
C02338=1182.826,-34.623,-43.198,179.702,5.741,149.107
C02339=1182.831,-34.872,-43.185,179.700,5.741,149.107
C02340=1182.836,-35.122,-43.173,179.698,5.741,149.108
C02341=1182.841,-35.371,-43.161,179.695,5.741,149.109
C02342=1182.847,-35.621,-43.149,179.693,5.740,149.109
C02343=1182.852,-35.870,-43.136,179.690,5.739,149.110
C02344=1182.857,-36.120,-43.124,179.688,5.739,149.111
C02345=1182.862,-36.370,-43.112,179.686,5.739,149.111
C02346=1182.867,-36.619,-43.100,179.683,5.738,149.112
C02347=1182.872,-36.870,-43.088,179.681,5.738,149.113
C02348=1182.877,-37.119,-43.075,179.678,5.738,149.113
C02349=1182.882,-37.369,-43.064,179.676,5.737,149.114
C02350=1182.887,-37.618,-43.051,179.674,5.737,149.114
C02351=1182.893,-37.868,-43.039,179.671,5.737,149.115
C02352=1182.898,-38.118,-43.026,179.669,5.736,149.116
C02353=1182.903,-38.367,-43.015,179.666,5.735,149.116
C02354=1182.908,-38.617,-43.003,179.664,5.735,149.117
C02355=1182.913,-38.867,-42.991,179.662,5.735,149.117
C02356=1182.919,-39.117,-42.979,179.659,5.734,149.118
C02357=1182.924,-39.366,-42.966,179.657,5.734,149.119
C02358=1182.929,-39.616,-42.954,179.654,5.734,149.120
C02359=1182.934,-39.865,-42.943,179.652,5.734,149.120
C02360=1182.939,-40.115,-42.930,179.650,5.733,149.121
C02361=1182.945,-40.365,-42.919,179.647,5.733,149.121
C02362=1182.950,-40.615,-42.907,179.645,5.732,149.122
C02363=1182.955,-40.864,-42.894,179.642,5.731,149.123
C02364=1182.960,-41.114,-42.883,179.640,5.732,149.123
C02365=1182.965,-41.363,-42.871,179.637,5.731,149.124
C02366=1182.970,-41.613,-42.858,179.635,5.731,149.124
C02367=1182.976,-41.863,-42.846,179.633,5.730,149.125
C02368=1182.980,-42.112,-42.835,179.631,5.730,149.126
C02369=1182.986,-42.362,-42.823,179.628,5.730,149.126
C02370=1182.991,-42.612,-42.811,179.626,5.729,149.127
C02371=1182.997,-42.861,-42.799,179.623,5.729,149.128
C02372=1183.002,-43.110,-42.788,179.621,5.728,149.128
C02373=1183.007,-43.360,-42.776,179.619,5.728,149.129
C02374=1183.012,-43.610,-42.763,179.616,5.728,149.130
C02375=1183.018,-43.860,-42.751,179.613,5.727,149.130
C02376=1183.022,-44.109,-42.740,179.611,5.727,149.131
C02377=1183.028,-44.359,-42.728,179.609,5.727,149.131
C02378=1183.033,-44.609,-42.716,179.606,5.727,149.132
C02379=1183.038,-44.858,-42.704,179.604,5.726,149.133
C02380=1183.043,-45.108,-42.692,179.602,5.725,149.133
C02381=1183.048,-45.358,-42.681,179.600,5.726,149.134
C02382=1183.053,-45.608,-42.669,179.597,5.725,149.135
C02383=1183.058,-45.857,-42.657,179.595,5.724,149.135
C02384=1183.064,-46.107,-42.645,179.592,5.724,149.136
C02385=1183.069,-46.356,-42.634,179.590,5.724,149.137
C02386=1183.074,-46.606,-42.622,179.588,5.724,149.137
C02387=1183.080,-46.856,-42.610,179.585,5.723,149.138
C02388=1183.085,-47.105,-42.599,179.582,5.723,149.139
C02389=1183.090,-47.355,-42.587,179.581,5.723,149.139
C02390=1183.095,-47.605,-42.574,179.578,5.722,149.140
C02391=1183.100,-47.854,-42.563,179.576,5.722,149.140
C02392=1183.105,-48.104,-42.551,179.573,5.721,149.141
C02393=1183.111,-48.354,-42.539,179.571,5.721,149.142
C02394=1183.116,-48.603,-42.528,179.569,5.721,149.142
C02395=1183.121,-48.853,-42.516,179.566,5.720,149.143
C02396=1183.126,-49.103,-42.505,179.564,5.720,149.143
C02397=1183.132,-49.373,-42.492,179.561,5.719,149.144
C02398=1183.138,-49.644,-42.480,179.559,5.720,149.145
C02399=1183.143,-49.914,-42.467,179.556,5.719,149.146
C02400=1183.148,-50.184,-42.454,179.554,5.719,149.146
C02401=1183.154,-50.434,-42.443,179.551,5.718,149.147
C02402=1183.160,-50.683,-42.431,179.549,5.717,149.147
C02403=1183.164,-50.933,-42.420,179.547,5.718,149.148
C02404=1183.170,-51.183,-42.408,179.544,5.717,149.149
C02405=1183.175,-51.432,-42.397,179.542,5.717,149.149
C02406=1183.180,-51.682,-42.385,179.539,5.716,149.150
C02407=1183.185,-51.932,-42.373,179.537,5.717,149.151
C02408=1183.191,-52.181,-42.362,179.535,5.716,149.151
C02409=1183.195,-52.431,-42.351,179.532,5.715,149.152
C02410=1183.201,-52.681,-42.339,179.530,5.715,149.153
C02411=1183.206,-52.931,-42.327,179.528,5.715,149.153
C02412=1183.211,-53.180,-42.315,179.525,5.714,149.154
C02413=1183.217,-53.429,-42.304,179.523,5.714,149.155
C02414=1183.222,-53.679,-42.293,179.521,5.714,149.155
C02415=1183.227,-53.929,-42.281,179.518,5.714,149.156
C02416=1183.232,-54.179,-42.270,179.516,5.713,149.156
C02417=1183.237,-54.429,-42.258,179.513,5.713,149.157
C02418=1183.242,-54.679,-42.247,179.512,5.713,149.158
C02419=1183.247,-54.928,-42.236,179.509,5.712,149.158
C02420=1183.253,-55.178,-42.224,179.506,5.712,149.159
C02421=1183.258,-55.427,-42.213,179.505,5.712,149.159
C02422=1183.263,-55.677,-42.201,179.502,5.711,149.160
C02423=1183.268,-55.926,-42.190,179.499,5.711,149.161
C02424=1183.274,-56.176,-42.178,179.497,5.710,149.161
C02425=1183.278,-56.426,-42.167,179.495,5.711,149.162
C02426=1183.284,-56.676,-42.156,179.492,5.710,149.163
C02427=1183.289,-56.926,-42.145,179.490,5.709,149.163
C02428=1183.295,-57.175,-42.133,179.488,5.710,149.164
C02429=1183.300,-57.425,-42.122,179.485,5.709,149.165
C02430=1183.304,-57.674,-42.110,179.483,5.708,149.165
C02431=1183.310,-57.924,-42.099,179.481,5.708,149.166
C02432=1183.315,-58.174,-42.088,179.479,5.708,149.167
C02433=1183.321,-58.424,-42.076,179.476,5.708,149.167
C02434=1183.325,-58.673,-42.065,179.474,5.707,149.168
C02435=1183.330,-58.923,-42.054,179.472,5.708,149.168
C02436=1183.336,-59.172,-42.042,179.469,5.707,149.169
C02437=1183.341,-59.423,-42.032,179.467,5.706,149.170
C02438=1183.347,-59.672,-42.020,179.465,5.707,149.170
C02439=1183.352,-59.921,-42.009,179.462,5.706,149.171
C02440=1183.357,-60.171,-41.998,179.460,5.705,149.171
C02441=1183.362,-60.422,-41.986,179.457,5.705,149.172
C02442=1183.367,-60.671,-41.975,179.455,5.705,149.173
C02443=1183.372,-60.920,-41.964,179.453,5.705,149.173
C02444=1183.378,-61.170,-41.952,179.450,5.704,149.174
C02445=1183.383,-61.420,-41.942,179.448,5.705,149.175
C02446=1183.388,-61.669,-41.931,179.446,5.704,149.175
C02447=1183.393,-61.919,-41.919,179.443,5.703,149.176
C02448=1183.398,-62.169,-41.908,179.441,5.704,149.177
C02449=1183.404,-62.418,-41.898,179.439,5.703,149.177
C02450=1183.409,-62.668,-41.886,179.436,5.702,149.178
C02451=1183.414,-62.919,-41.875,179.434,5.702,149.179
C02452=1183.419,-63.167,-41.864,179.432,5.702,149.179
C02453=1183.425,-63.417,-41.852,179.429,5.702,149.180
C02454=1183.430,-63.668,-41.842,179.427,5.701,149.180
C02455=1183.435,-63.917,-41.831,179.425,5.701,149.181
C02456=1183.440,-64.166,-41.819,179.422,5.701,149.182
C02457=1183.446,-64.417,-41.808,179.420,5.700,149.182
C02458=1183.451,-64.666,-41.797,179.418,5.700,149.183
C02459=1183.456,-64.915,-41.786,179.416,5.700,149.184
C02460=1183.461,-65.166,-41.775,179.413,5.699,149.184
C02461=1183.467,-65.415,-41.764,179.411,5.699,149.185
C02462=1183.472,-65.665,-41.753,179.409,5.699,149.185
C02463=1183.476,-65.915,-41.742,179.406,5.699,149.186
C02464=1183.482,-66.164,-41.731,179.404,5.699,149.187
C02465=1183.487,-66.414,-41.720,179.402,5.698,149.187
C02466=1183.493,-66.663,-41.709,179.399,5.698,149.188
C02467=1183.498,-66.913,-41.699,179.397,5.698,149.188
C02468=1183.503,-67.163,-41.687,179.395,5.697,149.189
C02469=1183.509,-67.413,-41.676,179.392,5.697,149.190
C02470=1183.513,-67.662,-41.665,179.390,5.697,149.190
C02471=1183.519,-67.912,-41.655,179.388,5.697,149.191
C02472=1183.524,-68.162,-41.644,179.385,5.696,149.192
C02473=1183.529,-68.412,-41.632,179.384,5.696,149.192
C02474=1183.535,-68.661,-41.622,179.381,5.696,149.193
C02475=1183.539,-68.911,-41.610,179.378,5.695,149.194
C02476=1183.545,-69.160,-41.600,179.377,5.695,149.194
C02477=1183.550,-69.410,-41.589,179.374,5.695,149.195
C02478=1183.555,-69.660,-41.578,179.371,5.694,149.196
C02479=1183.561,-69.910,-41.567,179.370,5.694,149.196
C02480=1183.566,-70.160,-41.556,179.367,5.694,149.197
C02481=1183.571,-70.409,-41.546,179.364,5.694,149.197
C02482=1183.576,-70.659,-41.535,179.363,5.694,149.198
C02483=1183.582,-70.908,-41.524,179.360,5.693,149.199
C02484=1183.587,-71.158,-41.512,179.357,5.693,149.199
C02485=1183.592,-71.408,-41.502,179.356,5.693,149.200
C02486=1183.597,-71.657,-41.491,179.353,5.692,149.201
C02487=1183.602,-71.908,-41.480,179.350,5.692,149.201
C02488=1183.608,-72.157,-41.470,179.349,5.692,149.202
C02489=1183.613,-72.407,-41.459,179.346,5.691,149.202
C02490=1183.618,-72.656,-41.449,179.344,5.691,149.203
C02491=1183.624,-72.906,-41.437,179.342,5.691,149.204
C02492=1183.629,-73.156,-41.427,179.339,5.691,149.204
C02493=1183.634,-73.406,-41.416,179.338,5.691,149.205
C02494=1183.639,-73.655,-41.405,179.335,5.690,149.206
C02495=1183.644,-73.905,-41.395,179.332,5.690,149.206
C02496=1183.650,-74.155,-41.384,179.331,5.690,149.207
C02497=1183.655,-74.404,-41.373,179.328,5.689,149.207
C02498=1183.660,-74.654,-41.363,179.325,5.689,149.208
C02499=1183.665,-74.904,-41.352,179.324,5.689,149.209
C02500=1183.671,-75.153,-41.341,179.321,5.689,149.209
C02501=1183.677,-75.425,-41.330,179.318,5.688,149.210
C02502=1183.682,-75.696,-41.318,179.316,5.688,149.211
C02503=1183.688,-75.966,-41.307,179.314,5.688,149.211
C02504=1183.694,-76.237,-41.295,179.311,5.687,149.212
C02505=1183.699,-76.487,-41.285,179.309,5.687,149.213
C02506=1183.704,-76.737,-41.274,179.307,5.687,149.213
C02507=1183.710,-76.987,-41.264,179.305,5.687,149.214
C02508=1183.714,-77.236,-41.252,179.302,5.686,149.215
C02509=1183.720,-77.486,-41.242,179.300,5.687,149.215
C02510=1183.725,-77.736,-41.232,179.298,5.686,149.216
C02511=1183.731,-77.986,-41.221,179.296,5.686,149.216
C02512=1183.735,-78.235,-41.210,179.293,5.685,149.217
C02513=1183.741,-78.485,-41.200,179.291,5.685,149.218
C02514=1183.746,-78.735,-41.189,179.289,5.685,149.218
C02515=1183.752,-78.984,-41.179,179.286,5.684,149.219
C02516=1183.756,-79.234,-41.168,179.284,5.684,149.220
C02517=1183.762,-79.484,-41.158,179.282,5.684,149.220
C02518=1183.767,-79.733,-41.147,179.279,5.684,149.221
C02519=1183.772,-79.983,-41.137,179.277,5.684,149.221
C02520=1183.778,-80.233,-41.127,179.275,5.684,149.222
C02521=1183.783,-80.483,-41.115,179.273,5.683,149.223
C02522=1183.788,-80.732,-41.105,179.270,5.683,149.223
C02523=1183.793,-80.982,-41.095,179.268,5.682,149.224
C02524=1183.799,-81.232,-41.084,179.266,5.682,149.225
C02525=1183.805,-81.481,-41.074,179.263,5.682,149.225
C02526=1183.810,-81.732,-41.064,179.261,5.682,149.226
C02527=1183.815,-81.981,-41.053,179.259,5.682,149.226
C02528=1183.820,-82.231,-41.042,179.257,5.682,149.227
C02529=1183.825,-82.480,-41.032,179.254,5.681,149.228
C02530=1183.830,-82.730,-41.022,179.252,5.681,149.228
C02531=1183.835,-82.980,-41.012,179.250,5.680,149.229
C02532=1183.841,-83.229,-41.002,179.248,5.681,149.230
C02533=1183.846,-83.480,-40.991,179.245,5.680,149.230
C02534=1183.851,-83.729,-40.981,179.243,5.680,149.231
C02535=1183.857,-83.979,-40.971,179.241,5.680,149.231
C02536=1183.862,-84.229,-40.960,179.238,5.680,149.232
C02537=1183.868,-84.479,-40.950,179.236,5.679,149.233
C02538=1183.873,-84.729,-40.939,179.234,5.679,149.233
C02539=1183.877,-84.977,-40.929,179.232,5.678,149.234
C02540=1183.883,-85.227,-40.919,179.230,5.679,149.235
C02541=1183.888,-85.477,-40.908,179.227,5.678,149.235
C02542=1183.893,-85.727,-40.898,179.225,5.678,149.236
C02543=1183.899,-85.976,-40.888,179.223,5.678,149.236
C02544=1183.904,-86.227,-40.877,179.221,5.677,149.237
C02545=1183.909,-86.476,-40.867,179.219,5.678,149.238
C02546=1183.914,-86.726,-40.857,179.216,5.677,149.238
C02547=1183.919,-86.976,-40.847,179.214,5.676,149.239
C02548=1183.925,-87.225,-40.836,179.212,5.677,149.240
C02549=1183.930,-87.475,-40.826,179.209,5.676,149.240
C02550=1183.936,-87.725,-40.816,179.207,5.676,149.241
C02551=1183.940,-87.974,-40.806,179.205,5.676,149.241
C02552=1183.945,-88.224,-40.795,179.203,5.676,149.242
C02553=1183.951,-88.474,-40.785,179.200,5.676,149.243
C02554=1183.957,-88.724,-40.776,179.198,5.675,149.243
C02555=1183.962,-88.974,-40.765,179.196,5.675,149.244
C02556=1183.967,-89.224,-40.756,179.194,5.675,149.245
C02557=1183.972,-89.473,-40.745,179.192,5.675,149.245
C02558=1183.978,-89.723,-40.735,179.189,5.674,149.246
C02559=1183.983,-89.973,-40.725,179.187,5.674,149.246
C02560=1183.988,-90.222,-40.715,179.185,5.674,149.247
C02561=1183.994,-90.472,-40.705,179.182,5.674,149.248
C02562=1183.999,-90.722,-40.694,179.181,5.674,149.248
C02563=1184.004,-90.971,-40.684,179.178,5.673,149.249
C02564=1184.009,-91.221,-40.674,179.175,5.673,149.250
C02565=1184.014,-91.472,-40.665,179.174,5.673,149.250
C02566=1184.020,-91.721,-40.654,179.171,5.672,149.251
C02567=1184.025,-91.971,-40.644,179.170,5.672,149.251
C02568=1184.030,-92.220,-40.634,179.167,5.672,149.252
C02569=1184.035,-92.470,-40.624,179.165,5.672,149.252
C02570=1184.041,-92.720,-40.614,179.163,5.672,149.253
C02571=1184.046,-92.969,-40.604,179.160,5.671,149.254
C02572=1184.052,-93.219,-40.595,179.158,5.671,149.254
C02573=1184.057,-93.469,-40.584,179.156,5.671,149.255
C02574=1184.062,-93.719,-40.574,179.154,5.671,149.255
C02575=1184.067,-93.968,-40.564,179.151,5.670,149.256
C02576=1184.073,-94.218,-40.554,179.149,5.671,149.257
C02577=1184.078,-94.468,-40.544,179.147,5.670,149.257
C02578=1184.083,-94.718,-40.535,179.144,5.670,149.258
C02579=1184.089,-94.967,-40.524,179.143,5.670,149.259
C02580=1184.094,-95.217,-40.514,179.140,5.669,149.259
C02581=1184.099,-95.467,-40.505,179.138,5.670,149.260
C02582=1184.104,-95.717,-40.495,179.136,5.669,149.260
C02583=1184.110,-95.966,-40.484,179.134,5.669,149.261
C02584=1184.115,-96.216,-40.475,179.132,5.668,149.262
C02585=1184.121,-96.466,-40.465,179.129,5.668,149.262
C02586=1184.126,-96.716,-40.455,179.127,5.668,149.263
C02587=1184.130,-96.965,-40.445,179.125,5.668,149.264
C02588=1184.136,-97.215,-40.435,179.123,5.668,149.264
C02589=1184.142,-97.465,-40.425,179.120,5.667,149.265
C02590=1184.147,-97.714,-40.416,179.118,5.668,149.265
C02591=1184.152,-97.965,-40.405,179.116,5.667,149.266
C02592=1184.157,-98.214,-40.396,179.114,5.667,149.267
C02593=1184.163,-98.464,-40.386,179.112,5.666,149.267
C02594=1184.168,-98.713,-40.376,179.109,5.666,149.268
C02595=1184.173,-98.963,-40.367,179.107,5.666,149.269
C02596=1184.178,-99.214,-40.356,179.105,5.666,149.269
C02597=1184.183,-99.463,-40.347,179.103,5.666,149.270
C02598=1184.189,-99.713,-40.337,179.101,5.665,149.270
C02599=1184.195,-99.962,-40.327,179.099,5.666,149.271
C02600=1184.200,-100.212,-40.318,179.096,5.665,149.271
C02601=1184.206,-100.462,-40.308,179.094,5.665,149.272
C02602=1184.210,-100.712,-40.298,179.092,5.665,149.273
C02603=1184.215,-100.961,-40.288,179.089,5.664,149.273
C02604=1184.221,-101.211,-40.279,179.087,5.665,149.274
C02605=1184.226,-101.483,-40.267,179.085,5.664,149.275
C02606=1184.232,-101.755,-40.257,179.083,5.664,149.275
C02607=1184.238,-102.026,-40.247,179.080,5.664,149.276
C02608=1184.243,-102.297,-40.236,179.078,5.663,149.277
C02609=1184.249,-102.547,-40.227,179.076,5.663,149.277
C02610=1184.254,-102.797,-40.217,179.073,5.663,149.278
C02611=1184.260,-103.047,-40.208,179.072,5.663,149.278
C02612=1184.264,-103.297,-40.198,179.069,5.663,149.279
C02613=1184.270,-103.547,-40.188,179.066,5.662,149.280
C02614=1184.275,-103.796,-40.179,179.065,5.662,149.280
C02615=1184.281,-104.046,-40.169,179.062,5.662,149.281
C02616=1184.286,-104.296,-40.160,179.061,5.662,149.282
C02617=1184.292,-104.546,-40.150,179.058,5.661,149.282
C02618=1184.296,-104.795,-40.140,179.056,5.661,149.283
C02619=1184.302,-105.045,-40.131,179.054,5.661,149.283
C02620=1184.307,-105.295,-40.121,179.052,5.661,149.284
C02621=1184.313,-105.545,-40.112,179.049,5.661,149.285
C02622=1184.317,-105.794,-40.102,179.048,5.661,149.285
C02623=1184.323,-106.045,-40.092,179.045,5.660,149.286
C02624=1184.328,-106.294,-40.083,179.043,5.661,149.287
C02625=1184.334,-106.544,-40.073,179.041,5.660,149.287
C02626=1184.339,-106.793,-40.064,179.038,5.660,149.288
C02627=1184.344,-107.043,-40.055,179.037,5.660,149.288
C02628=1184.350,-107.293,-40.045,179.034,5.659,149.289
C02629=1184.355,-107.542,-40.036,179.032,5.659,149.289
C02630=1184.360,-107.792,-40.025,179.030,5.659,149.290
C02631=1184.366,-108.042,-40.017,179.028,5.659,149.291
C02632=1184.371,-108.293,-40.007,179.025,5.658,149.291
C02633=1184.376,-108.542,-39.997,179.024,5.658,149.292
C02634=1184.381,-108.792,-39.988,179.021,5.658,149.293
C02635=1184.387,-109.041,-39.978,179.019,5.658,149.293
C02636=1184.392,-109.291,-39.969,179.017,5.658,149.294
C02637=1184.398,-109.541,-39.960,179.015,5.658,149.294
C02638=1184.402,-109.791,-39.950,179.012,5.657,149.295
C02639=1184.408,-110.040,-39.941,179.011,5.657,149.295
C02640=1184.413,-110.290,-39.931,179.008,5.657,149.296
C02641=1184.418,-110.540,-39.922,179.006,5.657,149.297
C02642=1184.424,-110.790,-39.913,179.004,5.657,149.297
C02643=1184.429,-111.039,-39.903,179.002,5.657,149.298
C02644=1184.434,-111.289,-39.894,179.000,5.656,149.299
C02645=1184.440,-111.539,-39.884,178.998,5.657,149.299
C02646=1184.445,-111.788,-39.875,178.995,5.656,149.300
C02647=1184.450,-112.038,-39.866,178.993,5.656,149.300
C02648=1184.456,-112.288,-39.856,178.991,5.655,149.301
C02649=1184.461,-112.538,-39.847,178.988,5.655,149.302
C02650=1184.466,-112.788,-39.838,178.987,5.655,149.302
C02651=1184.472,-113.038,-39.828,178.984,5.655,149.303
C02652=1184.477,-113.287,-39.819,178.983,5.655,149.303
C02653=1184.482,-113.537,-39.810,178.980,5.654,149.304
C02654=1184.488,-113.787,-39.800,178.978,5.654,149.305
C02655=1184.493,-114.037,-39.792,178.976,5.654,149.305
C02656=1184.498,-114.286,-39.782,178.974,5.654,149.306
C02657=1184.503,-114.536,-39.773,178.971,5.654,149.306
C02658=1184.509,-114.786,-39.764,178.970,5.654,149.307
C02659=1184.514,-115.036,-39.755,178.967,5.653,149.308
C02660=1184.519,-115.285,-39.745,178.965,5.653,149.308
C02661=1184.525,-115.535,-39.736,178.963,5.653,149.309
C02662=1184.530,-115.785,-39.727,178.961,5.653,149.309
C02663=1184.535,-116.035,-39.718,178.958,5.652,149.310
C02664=1184.540,-116.284,-39.708,178.957,5.652,149.311
C02665=1184.546,-116.534,-39.699,178.954,5.652,149.311
C02666=1184.551,-116.784,-39.690,178.953,5.652,149.312
C02667=1184.556,-117.034,-39.681,178.950,5.652,149.312
C02668=1184.562,-117.284,-39.672,178.948,5.652,149.313
C02669=1184.568,-117.534,-39.662,178.946,5.651,149.314
C02670=1184.573,-117.783,-39.653,178.944,5.651,149.314
C02671=1184.578,-118.032,-39.644,178.941,5.651,149.315
C02672=1184.583,-118.282,-39.635,178.940,5.651,149.315
C02673=1184.589,-118.533,-39.626,178.937,5.651,149.316
C02674=1184.594,-118.782,-39.617,178.935,5.651,149.317
C02675=1184.600,-119.032,-39.608,178.933,5.650,149.317
C02676=1184.604,-119.281,-39.599,178.931,5.650,149.318
C02677=1184.610,-119.531,-39.590,178.929,5.650,149.318
C02678=1184.616,-119.781,-39.580,178.927,5.650,149.319
C02679=1184.621,-120.031,-39.571,178.925,5.649,149.319
C02680=1184.626,-120.281,-39.562,178.923,5.650,149.320
C02681=1184.631,-120.531,-39.553,178.920,5.649,149.321
C02682=1184.636,-120.781,-39.545,178.918,5.649,149.321
C02683=1184.643,-121.030,-39.535,178.916,5.648,149.322
C02684=1184.648,-121.280,-39.527,178.914,5.649,149.323
C02685=1184.653,-121.529,-39.517,178.912,5.648,149.323
C02686=1184.658,-121.779,-39.508,178.910,5.648,149.324
C02687=1184.663,-122.029,-39.499,178.908,5.648,149.324
C02688=1184.668,-122.279,-39.490,178.906,5.648,149.325
C02689=1184.673,-122.529,-39.481,178.904,5.648,149.325
C02690=1184.679,-122.779,-39.472,178.901,5.648,149.326
C02691=1184.684,-123.029,-39.463,178.900,5.648,149.327
C02692=1184.690,-123.278,-39.454,178.897,5.647,149.327
C02693=1184.695,-123.528,-39.445,178.895,5.647,149.328
C02694=1184.701,-123.778,-39.437,178.893,5.647,149.329
C02695=1184.706,-124.028,-39.428,178.891,5.647,149.329
C02696=1184.711,-124.277,-39.419,178.889,5.646,149.330
C02697=1184.716,-124.527,-39.410,178.887,5.647,149.330
C02698=1184.722,-124.777,-39.400,178.885,5.646,149.331
C02699=1184.728,-125.027,-39.392,178.883,5.646,149.331
C02700=1184.733,-125.276,-39.383,178.880,5.646,149.332
C02701=1184.738,-125.526,-39.374,178.878,5.646,149.333
C02702=1184.743,-125.776,-39.365,178.876,5.645,149.333
C02703=1184.748,-126.026,-39.356,178.874,5.646,149.334
C02704=1184.754,-126.276,-39.347,178.872,5.645,149.334
C02705=1184.759,-126.526,-39.338,178.870,5.645,149.335
C02706=1184.764,-126.775,-39.330,178.867,5.645,149.336
C02707=1184.770,-127.025,-39.321,178.866,5.645,149.336
C02708=1184.775,-127.275,-39.312,178.863,5.644,149.337
C02709=1184.354,-127.286,-39.352,178.860,5.648,149.339
C02710=1184.349,-127.036,-39.361,178.862,5.648,149.338
C02711=1184.344,-126.786,-39.369,178.864,5.649,149.337
C02712=1184.338,-126.537,-39.378,178.866,5.649,149.337
C02713=1184.333,-126.287,-39.387,178.868,5.648,149.336
C02714=1184.327,-126.037,-39.397,178.870,5.649,149.336
C02715=1184.322,-125.787,-39.405,178.872,5.648,149.335
C02716=1184.316,-125.538,-39.414,178.874,5.649,149.335
C02717=1184.311,-125.288,-39.423,178.876,5.649,149.334
C02718=1184.306,-125.038,-39.432,178.879,5.650,149.333
C02719=1184.301,-124.788,-39.441,178.881,5.649,149.333
C02720=1184.296,-124.538,-39.450,178.883,5.650,149.332
C02721=1184.290,-124.289,-39.458,178.884,5.650,149.332
C02722=1184.285,-124.039,-39.467,178.887,5.650,149.331
C02723=1184.280,-123.789,-39.476,178.889,5.650,149.330
C02724=1184.274,-123.539,-39.486,178.891,5.651,149.330
C02725=1184.269,-123.289,-39.494,178.893,5.651,149.329
C02726=1184.263,-123.039,-39.503,178.896,5.651,149.328
C02727=1184.258,-122.790,-39.512,178.897,5.651,149.328
C02728=1184.252,-122.540,-39.521,178.900,5.651,149.327
C02729=1184.247,-122.291,-39.530,178.902,5.651,149.327
C02730=1184.242,-122.041,-39.539,178.904,5.652,149.326
C02731=1184.237,-121.791,-39.547,178.906,5.652,149.326
C02732=1184.231,-121.541,-39.557,178.908,5.652,149.325
C02733=1184.226,-121.291,-39.566,178.910,5.652,149.324
C02734=1184.221,-121.041,-39.575,178.912,5.653,149.324
C02735=1184.215,-120.791,-39.584,178.914,5.652,149.323
C02736=1184.210,-120.541,-39.593,178.917,5.653,149.323
C02737=1184.205,-120.291,-39.601,178.919,5.653,149.322
C02738=1184.199,-120.043,-39.611,178.921,5.654,149.322
C02739=1184.194,-119.793,-39.620,178.923,5.653,149.321
C02740=1184.189,-119.543,-39.629,178.925,5.654,149.320
C02741=1184.183,-119.293,-39.638,178.927,5.654,149.320
C02742=1184.178,-119.043,-39.647,178.929,5.654,149.319
C02743=1184.172,-118.793,-39.656,178.932,5.654,149.318
C02744=1184.167,-118.543,-39.665,178.934,5.655,149.318
C02745=1184.162,-118.294,-39.675,178.936,5.654,149.317
C02746=1184.157,-118.044,-39.684,178.938,5.655,149.317
C02747=1184.151,-117.794,-39.693,178.940,5.655,149.316
C02748=1184.146,-117.544,-39.702,178.942,5.655,149.315
C02749=1184.141,-117.294,-39.711,178.944,5.655,149.315
C02750=1184.136,-117.044,-39.720,178.947,5.656,149.314
C02751=1184.131,-116.795,-39.730,178.949,5.655,149.314
C02752=1184.124,-116.546,-39.739,178.951,5.656,149.313
C02753=1184.119,-116.296,-39.748,178.953,5.656,149.312
C02754=1184.114,-116.046,-39.757,178.955,5.656,149.312
C02755=1184.108,-115.796,-39.766,178.957,5.656,149.311
C02756=1184.103,-115.547,-39.776,178.959,5.657,149.311
C02757=1184.098,-115.297,-39.785,178.962,5.656,149.310
C02758=1184.093,-115.047,-39.793,178.964,5.657,149.309
C02759=1184.087,-114.797,-39.803,178.965,5.657,149.309
C02760=1184.082,-114.547,-39.813,178.968,5.658,149.308
C02761=1184.077,-114.298,-39.821,178.970,5.658,149.308
C02762=1184.071,-114.047,-39.831,178.972,5.658,149.307
C02763=1184.066,-113.798,-39.840,178.974,5.658,149.307
C02764=1184.061,-113.548,-39.849,178.977,5.658,149.306
C02765=1184.056,-113.299,-39.858,178.979,5.658,149.305
C02766=1184.050,-113.048,-39.868,178.981,5.659,149.305
C02767=1184.045,-112.799,-39.877,178.983,5.658,149.304
C02768=1184.040,-112.549,-39.886,178.985,5.659,149.303
C02769=1184.034,-112.299,-39.896,178.987,5.659,149.303
C02770=1184.029,-112.049,-39.905,178.989,5.659,149.302
C02771=1184.024,-111.800,-39.914,178.991,5.659,149.302
C02772=1184.018,-111.550,-39.924,178.994,5.660,149.301
C02773=1184.013,-111.300,-39.933,178.996,5.659,149.300
C02774=1184.007,-111.050,-39.943,178.998,5.660,149.300
C02775=1184.002,-110.801,-39.952,179.000,5.660,149.299
C02776=1183.997,-110.551,-39.961,179.002,5.661,149.299
C02777=1183.992,-110.301,-39.971,179.004,5.660,149.298
C02778=1183.986,-110.051,-39.980,179.006,5.661,149.297
C02779=1183.981,-109.802,-39.989,179.009,5.660,149.297
C02780=1183.976,-109.552,-39.999,179.011,5.661,149.296
C02781=1183.970,-109.302,-40.008,179.013,5.661,149.296
C02782=1183.965,-109.053,-40.018,179.015,5.662,149.295
C02783=1183.960,-108.802,-40.027,179.017,5.661,149.294
C02784=1183.955,-108.552,-40.036,179.019,5.662,149.294
C02785=1183.949,-108.303,-40.046,179.022,5.662,149.293
C02786=1183.944,-108.053,-40.055,179.024,5.662,149.293
C02787=1183.939,-107.803,-40.066,179.026,5.663,149.292
C02788=1183.934,-107.553,-40.074,179.028,5.663,149.292
C02789=1183.929,-107.304,-40.084,179.031,5.663,149.291
C02790=1183.923,-107.054,-40.094,179.032,5.663,149.290
C02791=1183.918,-106.804,-40.102,179.035,5.664,149.290
C02792=1183.912,-106.555,-40.113,179.037,5.663,149.289
C02793=1183.907,-106.305,-40.122,179.039,5.664,149.288
C02794=1183.901,-106.055,-40.132,179.041,5.664,149.288
C02795=1183.896,-105.805,-40.141,179.043,5.664,149.287
C02796=1183.891,-105.556,-40.150,179.045,5.664,149.286
C02797=1183.886,-105.305,-40.160,179.048,5.665,149.286
C02798=1183.881,-105.056,-40.170,179.050,5.664,149.285
C02799=1183.875,-104.806,-40.179,179.052,5.665,149.285
C02800=1183.870,-104.557,-40.189,179.054,5.665,149.284
C02801=1183.864,-104.306,-40.198,179.056,5.665,149.284
C02802=1183.860,-104.057,-40.208,179.059,5.666,149.283
C02803=1183.854,-103.807,-40.217,179.060,5.666,149.282
C02804=1183.849,-103.558,-40.227,179.063,5.666,149.282
C02805=1183.843,-103.307,-40.237,179.065,5.666,149.281
C02806=1183.839,-103.058,-40.247,179.067,5.667,149.280
C02807=1183.833,-102.808,-40.257,179.069,5.666,149.280
C02808=1183.828,-102.558,-40.266,179.072,5.667,149.279
C02809=1183.822,-102.309,-40.276,179.074,5.667,149.279
C02810=1183.817,-102.037,-40.286,179.076,5.667,149.278
C02811=1183.811,-101.765,-40.296,179.079,5.668,149.277
C02812=1183.805,-101.494,-40.307,179.081,5.667,149.277
C02813=1183.799,-101.222,-40.318,179.083,5.668,149.276
C02814=1183.794,-100.973,-40.327,179.086,5.669,149.275
C02815=1183.788,-100.723,-40.337,179.088,5.668,149.275
C02816=1183.783,-100.473,-40.347,179.090,5.668,149.274
C02817=1183.778,-100.223,-40.356,179.092,5.668,149.274
C02818=1183.773,-99.973,-40.366,179.095,5.669,149.273
C02819=1183.768,-99.724,-40.376,179.096,5.669,149.272
C02820=1183.762,-99.474,-40.386,179.099,5.669,149.272
C02821=1183.757,-99.225,-40.395,179.101,5.670,149.271
C02822=1183.752,-98.974,-40.406,179.103,5.670,149.270
C02823=1183.746,-98.724,-40.415,179.105,5.670,149.270
C02824=1183.741,-98.475,-40.425,179.107,5.670,149.269
C02825=1183.736,-98.225,-40.435,179.110,5.670,149.269
C02826=1183.731,-97.975,-40.444,179.112,5.670,149.268
C02827=1183.726,-97.725,-40.455,179.114,5.671,149.267
C02828=1183.720,-97.476,-40.465,179.116,5.671,149.267
C02829=1183.715,-97.226,-40.474,179.119,5.671,149.266
C02830=1183.709,-96.976,-40.484,179.121,5.672,149.266
C02831=1183.704,-96.727,-40.494,179.123,5.672,149.265
C02832=1183.699,-96.477,-40.504,179.126,5.672,149.264
C02833=1183.693,-96.227,-40.514,179.127,5.672,149.264
C02834=1183.689,-95.977,-40.523,179.130,5.672,149.263
C02835=1183.683,-95.728,-40.533,179.131,5.672,149.263
C02836=1183.677,-95.478,-40.543,179.134,5.673,149.262
C02837=1183.673,-95.228,-40.553,179.136,5.674,149.261
C02838=1183.667,-94.978,-40.563,179.138,5.673,149.261
C02839=1183.662,-94.729,-40.573,179.141,5.674,149.260
C02840=1183.657,-94.479,-40.583,179.143,5.674,149.259
C02841=1183.651,-94.229,-40.593,179.145,5.674,149.259
C02842=1183.646,-93.979,-40.603,179.147,5.674,149.258
C02843=1183.640,-93.730,-40.613,179.150,5.674,149.258
C02844=1183.635,-93.480,-40.623,179.152,5.675,149.257
C02845=1183.630,-93.230,-40.633,179.154,5.675,149.256
C02846=1183.624,-92.980,-40.643,179.157,5.675,149.256
C02847=1183.620,-92.731,-40.652,179.158,5.675,149.255
C02848=1183.614,-92.481,-40.663,179.161,5.676,149.254
C02849=1183.609,-92.231,-40.673,179.162,5.676,149.254
C02850=1183.604,-91.982,-40.683,179.165,5.676,149.253
C02851=1183.599,-91.732,-40.693,179.168,5.676,149.253
C02852=1183.593,-91.482,-40.703,179.169,5.676,149.252
C02853=1183.588,-91.232,-40.713,179.172,5.677,149.251
C02854=1183.583,-90.982,-40.723,179.174,5.677,149.251
C02855=1183.577,-90.733,-40.733,179.176,5.677,149.250
C02856=1183.572,-90.483,-40.744,179.178,5.677,149.249
C02857=1183.567,-90.233,-40.754,179.181,5.678,149.249
C02858=1183.562,-89.984,-40.763,179.183,5.678,149.248
C02859=1183.556,-89.734,-40.774,179.185,5.678,149.248
C02860=1183.551,-89.484,-40.784,179.188,5.678,149.247
C02861=1183.545,-89.234,-40.794,179.190,5.678,149.246
C02862=1183.540,-88.984,-40.804,179.192,5.679,149.246
C02863=1183.535,-88.734,-40.814,179.195,5.679,149.245
C02864=1183.530,-88.485,-40.824,179.196,5.679,149.245
C02865=1183.524,-88.235,-40.834,179.199,5.680,149.244
C02866=1183.519,-87.985,-40.845,179.201,5.679,149.243
C02867=1183.514,-87.736,-40.854,179.203,5.680,149.243
C02868=1183.509,-87.486,-40.865,179.206,5.680,149.242
C02869=1183.504,-87.236,-40.875,179.207,5.680,149.242
C02870=1183.498,-86.987,-40.885,179.210,5.681,149.241
C02871=1183.493,-86.737,-40.896,179.212,5.680,149.240
C02872=1183.488,-86.487,-40.906,179.214,5.681,149.240
C02873=1183.483,-86.238,-40.916,179.217,5.682,149.239
C02874=1183.477,-85.988,-40.926,179.219,5.682,149.238
C02875=1183.472,-85.738,-40.937,179.221,5.682,149.238
C02876=1183.467,-85.488,-40.947,179.223,5.682,149.237
C02877=1183.462,-85.238,-40.957,179.225,5.682,149.237
C02878=1183.456,-84.988,-40.968,179.228,5.683,149.236
C02879=1183.451,-84.739,-40.977,179.230,5.683,149.235
C02880=1183.446,-84.489,-40.988,179.232,5.683,149.235
C02881=1183.440,-84.239,-40.998,179.234,5.683,149.234
C02882=1183.435,-83.990,-41.008,179.237,5.684,149.233
C02883=1183.430,-83.740,-41.019,179.239,5.684,149.233
C02884=1183.425,-83.491,-41.030,179.241,5.684,149.232
C02885=1183.420,-83.240,-41.040,179.244,5.684,149.232
C02886=1183.414,-82.991,-41.050,179.246,5.684,149.231
C02887=1183.408,-82.741,-41.061,179.248,5.685,149.230
C02888=1183.404,-82.491,-41.071,179.251,5.685,149.230
C02889=1183.399,-82.242,-41.081,179.253,5.685,149.229
C02890=1183.394,-81.992,-41.091,179.255,5.686,149.228
C02891=1183.388,-81.742,-41.102,179.257,5.685,149.228
C02892=1183.382,-81.493,-41.112,179.259,5.686,149.227
C02893=1183.378,-81.243,-41.123,179.262,5.686,149.227
C02894=1183.372,-80.993,-41.133,179.264,5.686,149.226
C02895=1183.367,-80.743,-41.144,179.266,5.687,149.225
C02896=1183.361,-80.494,-41.154,179.269,5.687,149.225
C02897=1183.356,-80.243,-41.165,179.271,5.687,149.224
C02898=1183.351,-79.994,-41.175,179.273,5.688,149.224
C02899=1183.346,-79.745,-41.186,179.275,5.687,149.223
C02900=1183.341,-79.495,-41.196,179.277,5.688,149.222
C02901=1183.335,-79.245,-41.207,179.280,5.688,149.222
C02902=1183.330,-78.995,-41.217,179.282,5.688,149.221
C02903=1183.324,-78.745,-41.227,179.284,5.689,149.220
C02904=1183.320,-78.496,-41.239,179.287,5.689,149.220
C02905=1183.314,-78.246,-41.249,179.289,5.689,149.219
C02906=1183.309,-77.996,-41.259,179.291,5.690,149.219
C02907=1183.303,-77.746,-41.270,179.293,5.689,149.218
C02908=1183.298,-77.497,-41.281,179.296,5.690,149.217
C02909=1183.293,-77.247,-41.291,179.298,5.690,149.217
C02910=1183.288,-76.998,-41.301,179.300,5.690,149.216
C02911=1183.283,-76.747,-41.312,179.302,5.691,149.215
C02912=1183.277,-76.498,-41.323,179.305,5.691,149.215
C02913=1183.272,-76.248,-41.333,179.307,5.691,149.214
C02914=1183.266,-75.977,-41.345,179.310,5.691,149.213
C02915=1183.261,-75.707,-41.356,179.312,5.692,149.213
C02916=1183.255,-75.435,-41.368,179.315,5.693,149.212
C02917=1183.249,-75.165,-41.379,179.317,5.692,149.211
C02918=1183.244,-74.915,-41.390,179.319,5.693,149.211
C02919=1183.238,-74.665,-41.400,179.322,5.693,149.210
C02920=1183.233,-74.415,-41.412,179.324,5.693,149.210
C02921=1183.228,-74.166,-41.422,179.326,5.693,149.209
C02922=1183.223,-73.916,-41.433,179.329,5.694,149.208
C02923=1183.218,-73.667,-41.443,179.331,5.694,149.208
C02924=1183.213,-73.416,-41.454,179.333,5.694,149.207
C02925=1183.207,-73.167,-41.465,179.335,5.695,149.206
C02926=1183.202,-72.917,-41.476,179.338,5.695,149.206
C02927=1183.197,-72.667,-41.486,179.340,5.695,149.205
C02928=1183.192,-72.418,-41.497,179.342,5.695,149.205
C02929=1183.186,-72.167,-41.508,179.344,5.695,149.204
C02930=1183.181,-71.918,-41.518,179.347,5.696,149.203
C02931=1183.176,-71.668,-41.530,179.349,5.696,149.203
C02932=1183.170,-71.419,-41.540,179.351,5.696,149.202
C02933=1183.166,-71.169,-41.551,179.354,5.697,149.201
C02934=1183.160,-70.920,-41.561,179.356,5.697,149.201
C02935=1183.155,-70.670,-41.573,179.358,5.697,149.200
C02936=1183.149,-70.420,-41.584,179.361,5.698,149.200
C02937=1183.144,-70.170,-41.594,179.363,5.698,149.199
C02938=1183.139,-69.920,-41.605,179.365,5.698,149.198
C02939=1183.134,-69.671,-41.616,179.367,5.699,149.198
C02940=1183.129,-69.421,-41.627,179.370,5.698,149.197
C02941=1183.123,-69.172,-41.637,179.372,5.699,149.196
C02942=1183.118,-68.922,-41.649,179.374,5.700,149.196
C02943=1183.112,-68.672,-41.659,179.376,5.699,149.195
C02944=1183.108,-68.422,-41.670,179.379,5.700,149.194
C02945=1183.103,-68.172,-41.681,179.381,5.700,149.194
C02946=1183.097,-67.923,-41.692,179.383,5.700,149.193
C02947=1183.092,-67.673,-41.703,179.386,5.700,149.192
C02948=1183.086,-67.424,-41.714,179.388,5.701,149.192
C02949=1183.081,-67.174,-41.725,179.390,5.701,149.191
C02950=1183.077,-66.924,-41.736,179.393,5.701,149.191
C02951=1183.071,-66.675,-41.747,179.395,5.702,149.190
C02952=1183.066,-66.424,-41.758,179.397,5.702,149.189
C02953=1183.060,-66.176,-41.769,179.400,5.702,149.189
C02954=1183.055,-65.925,-41.780,179.402,5.703,149.188
C02955=1183.050,-65.675,-41.791,179.404,5.703,149.187
C02956=1183.044,-65.426,-41.802,179.407,5.703,149.187
C02957=1183.040,-65.176,-41.813,179.409,5.704,149.186
C02958=1183.035,-64.927,-41.824,179.411,5.703,149.186
C02959=1183.029,-64.677,-41.835,179.414,5.704,149.185
C02960=1183.024,-64.427,-41.846,179.416,5.705,149.184
C02961=1183.019,-64.177,-41.857,179.418,5.704,149.184
C02962=1183.014,-63.928,-41.868,179.421,5.705,149.183
C02963=1183.008,-63.678,-41.880,179.423,5.705,149.183
C02964=1183.003,-63.428,-41.890,179.425,5.705,149.182
C02965=1182.998,-63.179,-41.901,179.428,5.706,149.181
C02966=1182.993,-62.929,-41.913,179.430,5.706,149.181
C02967=1182.988,-62.679,-41.924,179.433,5.707,149.180
C02968=1182.982,-62.430,-41.935,179.435,5.706,149.179
C02969=1182.977,-62.180,-41.946,179.437,5.707,149.179
C02970=1182.972,-61.929,-41.957,179.439,5.708,149.178
C02971=1182.967,-61.681,-41.968,179.442,5.707,149.177
C02972=1182.961,-61.431,-41.980,179.444,5.708,149.177
C02973=1182.956,-61.181,-41.991,179.446,5.708,149.176
C02974=1182.951,-60.931,-42.001,179.448,5.708,149.175
C02975=1182.945,-60.682,-42.013,179.451,5.709,149.175
C02976=1182.941,-60.432,-42.025,179.453,5.709,149.174
C02977=1182.935,-60.182,-42.035,179.455,5.709,149.174
C02978=1182.930,-59.932,-42.047,179.458,5.710,149.173
C02979=1182.925,-59.683,-42.058,179.460,5.710,149.172
C02980=1182.920,-59.433,-42.069,179.463,5.711,149.172
C02981=1182.914,-59.184,-42.081,179.465,5.711,149.171
C02982=1182.909,-58.934,-42.091,179.467,5.711,149.170
C02983=1182.904,-58.684,-42.103,179.470,5.711,149.170
C02984=1182.899,-58.434,-42.114,179.471,5.711,149.169
C02985=1182.894,-58.185,-42.125,179.474,5.712,149.169
C02986=1182.888,-57.935,-42.137,179.477,5.712,149.168
C02987=1182.883,-57.685,-42.148,179.479,5.713,149.167
C02988=1182.878,-57.435,-42.160,179.481,5.713,149.167
C02989=1182.873,-57.186,-42.171,179.484,5.713,149.166
C02990=1182.868,-56.937,-42.182,179.486,5.714,149.166
C02991=1182.863,-56.687,-42.194,179.488,5.714,149.165
C02992=1182.858,-56.436,-42.204,179.491,5.714,149.164
C02993=1182.852,-56.187,-42.216,179.493,5.715,149.164
C02994=1182.847,-55.937,-42.227,179.495,5.715,149.163
C02995=1182.841,-55.688,-42.239,179.498,5.715,149.162
C02996=1182.837,-55.438,-42.250,179.500,5.716,149.162
C02997=1182.831,-55.189,-42.262,179.502,5.716,149.161
C02998=1182.826,-54.939,-42.273,179.504,5.716,149.160
C02999=1182.821,-54.689,-42.285,179.507,5.716,149.160
C03000=1182.816,-54.440,-42.296,179.509,5.717,149.159
C03001=1182.811,-54.189,-42.307,179.512,5.717,149.158
C03002=1182.805,-53.940,-42.318,179.514,5.717,149.158
C03003=1182.800,-53.690,-42.330,179.516,5.718,149.157
C03004=1182.795,-53.440,-42.342,179.519,5.718,149.157
C03005=1182.790,-53.191,-42.353,179.521,5.718,149.156
C03006=1182.785,-52.941,-42.365,179.523,5.719,149.155
C03007=1182.779,-52.692,-42.376,179.526,5.719,149.155
C03008=1182.774,-52.442,-42.388,179.529,5.720,149.154
C03009=1182.768,-52.192,-42.400,179.530,5.720,149.154
C03010=1182.764,-51.942,-42.411,179.533,5.720,149.153
C03011=1182.758,-51.693,-42.423,179.535,5.720,149.152
C03012=1182.754,-51.443,-42.434,179.538,5.721,149.152
C03013=1182.748,-51.194,-42.445,179.540,5.721,149.151
C03014=1182.743,-50.944,-42.457,179.542,5.721,149.150
C03015=1182.738,-50.694,-42.469,179.545,5.722,149.150
C03016=1182.733,-50.445,-42.480,179.547,5.723,149.149
C03017=1182.727,-50.195,-42.492,179.549,5.722,149.148
C03018=1182.721,-49.925,-42.504,179.552,5.723,149.148
C03019=1182.716,-49.654,-42.517,179.555,5.723,149.147
C03020=1182.711,-49.384,-42.530,179.557,5.724,149.146
C03021=1182.705,-49.114,-42.542,179.560,5.724,149.146
C03022=1182.699,-48.864,-42.554,179.562,5.725,149.145
C03023=1182.695,-48.614,-42.565,179.564,5.724,149.144
C03024=1182.689,-48.364,-42.577,179.567,5.725,149.144
C03025=1182.684,-48.115,-42.589,179.569,5.726,149.143
C03026=1182.679,-47.865,-42.600,179.572,5.726,149.142
C03027=1182.674,-47.615,-42.612,179.574,5.726,149.142
C03028=1182.668,-47.366,-42.623,179.576,5.727,149.141
C03029=1182.663,-47.117,-42.636,179.579,5.727,149.141
C03030=1182.658,-46.867,-42.648,179.581,5.727,149.140
C03031=1182.653,-46.617,-42.659,179.583,5.727,149.139
C03032=1182.648,-46.367,-42.671,179.586,5.728,149.139
C03033=1182.642,-46.117,-42.683,179.588,5.728,149.138
C03034=1182.637,-45.868,-42.694,179.591,5.729,149.137
C03035=1182.632,-45.618,-42.706,179.593,5.729,149.137
C03036=1182.627,-45.368,-42.719,179.595,5.729,149.136
C03037=1182.622,-45.119,-42.730,179.598,5.730,149.135
C03038=1182.616,-44.870,-42.741,179.600,5.730,149.135
C03039=1182.611,-44.620,-42.753,179.602,5.730,149.134
C03040=1182.606,-44.370,-42.765,179.605,5.730,149.134
C03041=1182.601,-44.121,-42.777,179.607,5.731,149.133
C03042=1182.595,-43.871,-42.789,179.610,5.732,149.132
C03043=1182.590,-43.621,-42.801,179.612,5.731,149.132
C03044=1182.585,-43.371,-42.812,179.614,5.732,149.131
C03045=1182.580,-43.122,-42.825,179.617,5.733,149.131
C03046=1182.575,-42.872,-42.837,179.619,5.733,149.130
C03047=1182.570,-42.622,-42.848,179.622,5.734,149.129
C03048=1182.565,-42.372,-42.860,179.623,5.734,149.129
C03049=1182.560,-42.123,-42.873,179.626,5.734,149.128
C03050=1182.554,-41.873,-42.884,179.629,5.734,149.127
C03051=1182.549,-41.623,-42.896,179.631,5.735,149.127
C03052=1182.544,-41.374,-42.908,179.633,5.735,149.126
C03053=1182.539,-41.124,-42.920,179.636,5.735,149.125
C03054=1182.533,-40.874,-42.932,179.638,5.736,149.125
C03055=1182.529,-40.625,-42.943,179.641,5.737,149.124
C03056=1182.524,-40.375,-42.956,179.643,5.737,149.123
C03057=1182.518,-40.125,-42.968,179.645,5.737,149.123
C03058=1182.513,-39.875,-42.980,179.647,5.737,149.122
C03059=1182.508,-39.626,-42.992,179.650,5.738,149.122
C03060=1182.503,-39.376,-43.004,179.653,5.738,149.121
C03061=1182.498,-39.127,-43.016,179.654,5.738,149.120
C03062=1182.492,-38.877,-43.028,179.657,5.739,149.120
C03063=1182.487,-38.627,-43.040,179.660,5.739,149.119
C03064=1182.482,-38.378,-43.053,179.662,5.740,149.118
C03065=1182.476,-38.128,-43.064,179.665,5.740,149.118
C03066=1182.472,-37.878,-43.076,179.667,5.740,149.117
C03067=1182.467,-37.629,-43.088,179.669,5.741,149.116
C03068=1182.461,-37.379,-43.100,179.671,5.741,149.116
C03069=1182.456,-37.130,-43.113,179.674,5.742,149.115
C03070=1182.451,-36.880,-43.125,179.677,5.742,149.115
C03071=1182.446,-36.631,-43.137,179.678,5.742,149.114
C03072=1182.440,-36.381,-43.149,179.681,5.743,149.113
C03073=1182.435,-36.131,-43.161,179.684,5.743,149.113
C03074=1182.430,-35.882,-43.173,179.686,5.744,149.112
C03075=1182.425,-35.632,-43.185,179.689,5.744,149.112
C03076=1182.420,-35.382,-43.198,179.691,5.744,149.111
C03077=1182.414,-35.133,-43.210,179.693,5.745,149.110
C03078=1182.409,-34.883,-43.222,179.695,5.745,149.110
C03079=1182.404,-34.633,-43.234,179.698,5.746,149.109
C03080=1182.399,-34.384,-43.247,179.701,5.746,149.108
C03081=1182.393,-34.134,-43.258,179.702,5.746,149.108
C03082=1182.389,-33.884,-43.271,179.705,5.747,149.107
C03083=1182.383,-33.634,-43.283,179.708,5.747,149.106
C03084=1182.378,-33.385,-43.296,179.710,5.748,149.106
C03085=1182.373,-33.135,-43.309,179.713,5.748,149.105
C03086=1182.368,-32.886,-43.320,179.715,5.748,149.105
C03087=1182.363,-32.636,-43.332,179.717,5.749,149.104
C03088=1182.358,-32.387,-43.344,179.719,5.749,149.103
C03089=1182.353,-32.137,-43.357,179.722,5.750,149.103
C03090=1182.347,-31.887,-43.369,179.725,5.750,149.102
C03091=1182.342,-31.638,-43.381,179.727,5.751,149.101
C03092=1182.338,-31.388,-43.394,179.729,5.751,149.101
C03093=1182.332,-31.138,-43.406,179.732,5.751,149.100
C03094=1182.327,-30.889,-43.419,179.734,5.752,149.099
C03095=1182.322,-30.639,-43.431,179.737,5.752,149.099
C03096=1182.316,-30.389,-43.443,179.739,5.753,149.098
C03097=1182.311,-30.140,-43.456,179.742,5.753,149.098
C03098=1182.306,-29.890,-43.468,179.743,5.753,149.097
C03099=1182.301,-29.641,-43.480,179.746,5.754,149.096
C03100=1182.296,-29.391,-43.493,179.749,5.754,149.096
C03101=1182.291,-29.141,-43.505,179.751,5.755,149.095
C03102=1182.286,-28.892,-43.518,179.754,5.755,149.095
C03103=1182.281,-28.642,-43.530,179.756,5.756,149.094
C03104=1182.275,-28.392,-43.542,179.758,5.756,149.093
C03105=1182.269,-28.143,-43.556,179.761,5.756,149.093
C03106=1182.265,-27.893,-43.569,179.763,5.757,149.092
C03107=1182.260,-27.643,-43.581,179.766,5.757,149.091
C03108=1182.254,-27.393,-43.593,179.769,5.758,149.091
C03109=1182.249,-27.144,-43.606,179.771,5.759,149.090
C03110=1182.244,-26.895,-43.618,179.773,5.758,149.089
C03111=1182.239,-26.644,-43.630,179.775,5.759,149.089
C03112=1182.234,-26.395,-43.643,179.778,5.760,149.088
C03113=1182.229,-26.146,-43.656,179.780,5.760,149.088
C03114=1182.224,-25.896,-43.668,179.783,5.760,149.087
C03115=1182.219,-25.647,-43.681,179.786,5.761,149.086
C03116=1182.214,-25.396,-43.693,179.787,5.761,149.086
C03117=1182.208,-25.147,-43.706,179.790,5.761,149.085
C03118=1182.203,-24.897,-43.719,179.793,5.762,149.084
C03119=1182.198,-24.648,-43.732,179.795,5.763,149.084
C03120=1182.193,-24.399,-43.744,179.797,5.763,149.083
C03121=1182.188,-24.148,-43.756,179.800,5.764,149.082
C03122=1182.182,-23.879,-43.770,179.803,5.764,149.082
C03123=1182.176,-23.609,-43.784,179.805,5.764,149.081
C03124=1182.171,-23.339,-43.798,179.808,5.765,149.080
C03125=1182.165,-23.070,-43.812,179.810,5.766,149.080
C03126=1182.161,-22.820,-43.825,179.813,5.766,149.079
C03127=1182.155,-22.571,-43.837,179.815,5.767,149.078
C03128=1182.150,-22.321,-43.849,179.818,5.766,149.078
C03129=1182.145,-22.071,-43.862,179.820,5.767,149.077
C03130=1182.140,-21.821,-43.875,179.822,5.768,149.077
C03131=1182.134,-21.572,-43.888,179.825,5.768,149.076
C03132=1182.129,-21.322,-43.900,179.827,5.769,149.075
C03133=1182.124,-21.073,-43.913,179.830,5.769,149.075
C03134=1182.120,-20.823,-43.926,179.833,5.770,149.074
C03135=1182.114,-20.573,-43.939,179.835,5.769,149.073
C03136=1182.109,-20.324,-43.952,179.837,5.770,149.073
C03137=1182.104,-20.075,-43.964,179.839,5.771,149.072
C03138=1182.099,-19.825,-43.977,179.842,5.771,149.072
C03139=1182.093,-19.575,-43.990,179.844,5.772,149.071
C03140=1182.088,-19.326,-44.003,179.847,5.772,149.070
C03141=1182.084,-19.076,-44.016,179.850,5.773,149.070
C03142=1182.078,-18.826,-44.029,179.852,5.773,149.069
C03143=1182.073,-18.577,-44.042,179.854,5.773,149.068
C03144=1182.067,-18.328,-44.054,179.857,5.774,149.068
C03145=1182.063,-18.077,-44.067,179.859,5.774,149.067
C03146=1182.057,-17.828,-44.081,179.861,5.775,149.067
C03147=1182.052,-17.579,-44.093,179.864,5.776,149.066
C03148=1182.047,-17.329,-44.106,179.867,5.776,149.065
C03149=1182.042,-17.079,-44.119,179.869,5.776,149.065
C03150=1182.036,-16.830,-44.132,179.871,5.777,149.064
C03151=1182.032,-16.580,-44.145,179.874,5.778,149.063
C03152=1182.027,-16.330,-44.158,179.876,5.777,149.063
C03153=1182.021,-16.081,-44.171,179.878,5.778,149.062
C03154=1182.016,-15.831,-44.184,179.881,5.779,149.062
C03155=1182.011,-15.581,-44.196,179.884,5.779,149.061
C03156=1182.006,-15.331,-44.210,179.886,5.780,149.060
C03157=1182.001,-15.082,-44.222,179.889,5.780,149.060
C03158=1181.996,-14.833,-44.236,179.891,5.781,149.059
C03159=1181.991,-14.583,-44.249,179.894,5.781,149.058
C03160=1181.986,-14.333,-44.262,179.896,5.782,149.058
C03161=1181.981,-14.084,-44.275,179.899,5.783,149.057
C03162=1181.975,-13.834,-44.288,179.901,5.782,149.056
C03163=1181.970,-13.584,-44.301,179.903,5.783,149.056
C03164=1181.965,-13.334,-44.314,179.906,5.784,149.055
C03165=1181.960,-13.085,-44.328,179.908,5.784,149.055
C03166=1181.955,-12.836,-44.340,179.911,5.785,149.054
C03167=1181.950,-12.586,-44.354,179.913,5.785,149.053
C03168=1181.945,-12.336,-44.366,179.916,5.786,149.053
C03169=1181.939,-12.086,-44.380,179.918,5.786,149.052
C03170=1181.935,-11.837,-44.393,179.921,5.787,149.052
C03171=1181.929,-11.588,-44.406,179.923,5.788,149.051
C03172=1181.924,-11.338,-44.419,179.926,5.788,149.050
C03173=1181.919,-11.088,-44.432,179.929,5.789,149.050
C03174=1181.914,-10.839,-44.446,179.930,5.789,149.049
C03175=1181.909,-10.589,-44.459,179.933,5.789,149.048
C03176=1181.903,-10.340,-44.472,179.935,5.790,149.048
C03177=1181.899,-10.090,-44.485,179.938,5.790,149.047
C03178=1181.893,-9.841,-44.499,179.940,5.791,149.047
C03179=1181.888,-9.591,-44.512,179.943,5.791,149.046
C03180=1181.883,-9.341,-44.525,179.945,5.792,149.045
C03181=1181.878,-9.092,-44.539,179.948,5.793,149.045
C03182=1181.873,-8.842,-44.551,179.950,5.793,149.044
C03183=1181.868,-8.592,-44.565,179.953,5.794,149.043
C03184=1181.863,-8.343,-44.578,179.955,5.794,149.043
C03185=1181.858,-8.093,-44.592,179.958,5.795,149.042
C03186=1181.853,-7.844,-44.604,179.961,5.795,149.041
C03187=1181.848,-7.594,-44.619,179.963,5.796,149.041
C03188=1181.843,-7.345,-44.631,179.965,5.796,149.040
C03189=1181.837,-7.095,-44.644,179.967,5.796,149.040
C03190=1181.833,-6.846,-44.658,179.970,5.797,149.039
C03191=1181.827,-6.596,-44.671,179.972,5.798,149.038
C03192=1181.822,-6.346,-44.685,179.975,5.798,149.038
C03193=1181.817,-6.097,-44.698,179.978,5.798,149.037
C03194=1181.811,-5.847,-44.712,179.980,5.799,149.037
C03195=1181.807,-5.598,-44.725,179.982,5.800,149.036
C03196=1181.801,-5.348,-44.739,179.985,5.800,149.035
C03197=1181.797,-5.099,-44.752,179.987,5.801,149.035
C03198=1181.791,-4.849,-44.766,179.990,5.802,149.034
C03199=1181.786,-4.598,-44.779,179.993,5.802,149.033
C03200=1181.781,-4.349,-44.792,179.995,5.802,149.033
C03201=1181.776,-4.099,-44.806,179.997,5.803,149.032
C03202=1181.771,-3.850,-44.819,-180.000,5.804,149.032
C03203=1181.766,-3.600,-44.833,-179.997,5.804,149.031
C03204=1181.760,-3.351,-44.847,-179.995,5.805,149.030
C03205=1181.756,-3.101,-44.860,-179.992,5.806,149.030
C03206=1181.750,-2.852,-44.874,-179.990,5.806,149.029
C03207=1181.746,-2.602,-44.887,-179.988,5.807,149.029
C03208=1181.740,-2.353,-44.901,-179.986,5.807,149.028
C03209=1181.735,-2.103,-44.914,-179.983,5.807,149.027
C03210=1181.730,-1.854,-44.927,-179.980,5.808,149.026
C03211=1181.725,-1.604,-44.941,-179.978,5.808,149.026
C03212=1181.720,-1.354,-44.955,-179.975,5.809,149.025
C03213=1181.715,-1.105,-44.969,-179.973,5.809,149.025
C03214=1181.710,-0.855,-44.982,-179.971,5.810,149.024
C03215=1181.704,-0.606,-44.996,-179.968,5.811,149.023
C03216=1181.700,-0.356,-45.009,-179.965,5.811,149.023
C03217=1181.695,-0.106,-45.023,-179.963,5.812,149.022
C03218=1181.689,0.143,-45.037,-179.961,5.812,149.022
C03219=1181.685,0.393,-45.050,-179.958,5.813,149.021
C03220=1181.679,0.642,-45.064,-179.955,5.813,149.020
C03221=1181.674,0.892,-45.078,-179.953,5.814,149.020
C03222=1181.669,1.142,-45.092,-179.950,5.815,149.019
C03223=1181.664,1.391,-45.105,-179.948,5.815,149.018
C03224=1181.659,1.641,-45.119,-179.946,5.816,149.018
C03225=1181.653,1.890,-45.133,-179.943,5.816,149.017
C03226=1181.648,2.159,-45.148,-179.940,5.817,149.017
C03227=1181.642,2.429,-45.163,-179.938,5.817,149.016
C03228=1181.638,2.698,-45.177,-179.935,5.818,149.015
C03229=1181.632,2.967,-45.192,-179.932,5.819,149.015
C03230=1181.627,3.216,-45.206,-179.930,5.820,149.014
C03231=1181.621,3.467,-45.220,-179.927,5.820,149.013
C03232=1181.616,3.716,-45.233,-179.924,5.821,149.013
C03233=1181.612,3.965,-45.247,-179.922,5.822,149.012
C03234=1181.607,4.215,-45.261,-179.919,5.822,149.012
C03235=1181.601,4.464,-45.275,-179.917,5.823,149.011
C03236=1181.596,4.714,-45.289,-179.914,5.823,149.010
C03237=1181.591,4.964,-45.303,-179.912,5.824,149.010
C03238=1181.586,5.212,-45.317,-179.909,5.825,149.009
C03239=1181.581,5.463,-45.330,-179.907,5.825,149.008
C03240=1181.576,5.712,-45.344,-179.904,5.826,149.008
C03241=1181.570,5.961,-45.358,-179.902,5.826,149.007
C03242=1181.565,6.211,-45.373,-179.899,5.827,149.006
C03243=1181.560,6.461,-45.387,-179.897,5.828,149.006
C03244=1181.555,6.710,-45.399,-179.894,5.828,149.005
C03245=1181.550,6.960,-45.414,-179.892,5.829,149.005
C03246=1181.545,7.210,-45.428,-179.889,5.829,149.004
C03247=1181.540,7.459,-45.442,-179.887,5.830,149.004
C03248=1181.535,7.708,-45.456,-179.884,5.830,149.003
C03249=1181.530,7.958,-45.470,-179.882,5.831,149.002
C03250=1181.525,8.208,-45.485,-179.879,5.832,149.002
C03251=1181.520,8.457,-45.497,-179.877,5.832,149.001
C03252=1181.515,8.707,-45.512,-179.874,5.833,149.000
C03253=1181.510,8.957,-45.526,-179.872,5.834,149.000
C03254=1181.505,9.206,-45.540,-179.869,5.834,148.999
C03255=1181.499,9.455,-45.554,-179.867,5.834,148.998
C03256=1181.494,9.705,-45.568,-179.864,5.835,148.998
C03257=1181.490,9.955,-45.583,-179.862,5.836,148.997
C03258=1181.485,10.204,-45.597,-179.859,5.836,148.997
C03259=1181.479,10.453,-45.611,-179.857,5.837,148.996
C03260=1181.474,10.703,-45.625,-179.854,5.838,148.996
C03261=1181.469,10.953,-45.639,-179.852,5.838,148.995
C03262=1181.464,11.203,-45.654,-179.849,5.839,148.994
C03263=1181.459,11.452,-45.668,-179.847,5.839,148.994
C03264=1181.454,11.701,-45.682,-179.844,5.840,148.993
C03265=1181.449,11.951,-45.696,-179.842,5.840,148.992
C03266=1181.444,12.201,-45.710,-179.839,5.841,148.992
C03267=1181.439,12.450,-45.725,-179.837,5.842,148.991
C03268=1181.433,12.699,-45.739,-179.834,5.842,148.990
C03269=1181.428,12.949,-45.753,-179.832,5.843,148.990
C03270=1181.423,13.199,-45.767,-179.829,5.844,148.989
C03271=1181.418,13.449,-45.781,-179.827,5.844,148.989
C03272=1181.413,13.698,-45.795,-179.824,5.845,148.988
C03273=1181.408,13.947,-45.810,-179.821,5.846,148.988
C03274=1181.403,14.197,-45.824,-179.819,5.847,148.987
C03275=1181.398,14.447,-45.838,-179.816,5.848,148.986
C03276=1181.393,14.696,-45.852,-179.814,5.848,148.986
C03277=1181.388,14.946,-45.867,-179.811,5.848,148.985
C03278=1181.382,15.195,-45.881,-179.809,5.849,148.985
C03279=1181.378,15.445,-45.895,-179.806,5.850,148.984
C03280=1181.373,15.694,-45.910,-179.804,5.850,148.983
C03281=1181.368,15.944,-45.924,-179.801,5.851,148.983
C03282=1181.363,16.193,-45.938,-179.799,5.852,148.982
C03283=1181.358,16.443,-45.953,-179.796,5.852,148.981
C03284=1181.352,16.692,-45.967,-179.794,5.853,148.981
C03285=1181.348,16.942,-45.981,-179.791,5.853,148.980
C03286=1181.343,17.191,-45.996,-179.789,5.854,148.980
C03287=1181.338,17.441,-46.010,-179.786,5.854,148.979
C03288=1181.332,17.691,-46.025,-179.784,5.855,148.978
C03289=1181.327,17.940,-46.039,-179.781,5.856,148.978
C03290=1181.322,18.190,-46.054,-179.778,5.857,148.977
C03291=1181.318,18.439,-46.069,-179.776,5.858,148.977
C03292=1181.312,18.688,-46.082,-179.773,5.858,148.976
C03293=1181.307,18.938,-46.097,-179.771,5.859,148.975
C03294=1181.302,19.188,-46.111,-179.768,5.860,148.975
C03295=1181.297,19.437,-46.125,-179.766,5.860,148.974
C03296=1181.292,19.687,-46.141,-179.763,5.861,148.973
C03297=1181.287,19.936,-46.155,-179.761,5.862,148.973
C03298=1181.282,20.186,-46.169,-179.758,5.862,148.972
C03299=1181.277,20.435,-46.184,-179.756,5.863,148.972
C03300=1181.272,20.685,-46.199,-179.753,5.863,148.971
C03301=1181.267,20.935,-46.213,-179.751,5.864,148.970
C03302=1181.261,21.184,-46.228,-179.748,5.865,148.970
C03303=1181.256,21.433,-46.243,-179.745,5.866,148.969
C03304=1181.251,21.683,-46.257,-179.743,5.867,148.969
C03305=1181.247,21.932,-46.271,-179.740,5.867,148.968
C03306=1181.242,22.181,-46.286,-179.738,5.868,148.968
C03307=1181.236,22.432,-46.301,-179.735,5.868,148.967
C03308=1181.232,22.681,-46.316,-179.733,5.869,148.966
C03309=1181.227,22.930,-46.330,-179.731,5.870,148.966
C03310=1181.222,23.180,-46.344,-179.728,5.870,148.965
C03311=1181.216,23.429,-46.360,-179.725,5.871,148.964
C03312=1181.211,23.679,-46.374,-179.723,5.872,148.964
C03313=1181.206,23.929,-46.389,-179.720,5.873,148.963
C03314=1181.202,24.178,-46.404,-179.717,5.873,148.963
C03315=1181.196,24.428,-46.418,-179.715,5.874,148.962
C03316=1181.191,24.677,-46.433,-179.712,5.875,148.961
C03317=1181.186,24.927,-46.448,-179.710,5.875,148.961
C03318=1181.181,25.176,-46.463,-179.708,5.876,148.960
C03319=1181.176,25.426,-46.478,-179.705,5.877,148.960
C03320=1181.171,25.675,-46.493,-179.702,5.877,148.959
C03321=1181.166,25.925,-46.507,-179.700,5.878,148.958
C03322=1181.161,26.174,-46.522,-179.697,5.879,148.958
C03323=1181.156,26.424,-46.537,-179.694,5.880,148.957
C03324=1181.151,26.673,-46.552,-179.692,5.881,148.957
C03325=1181.146,26.923,-46.567,-179.689,5.881,148.956
C03326=1181.141,27.172,-46.582,-179.687,5.882,148.956
C03327=1181.136,27.422,-46.596,-179.685,5.882,148.955
C03328=1181.131,27.671,-46.611,-179.682,5.883,148.954
C03329=1181.126,27.921,-46.626,-179.680,5.884,148.954
C03330=1181.120,28.190,-46.642,-179.677,5.885,148.953
C03331=1181.115,28.459,-46.658,-179.674,5.886,148.952
C03332=1181.110,28.727,-46.674,-179.671,5.886,148.952
C03333=1181.104,28.996,-46.690,-179.668,5.887,148.951
C03334=1181.099,29.246,-46.705,-179.665,5.888,148.950
C03335=1181.094,29.495,-46.720,-179.663,5.889,148.950
C03336=1181.089,29.744,-46.735,-179.661,5.889,148.949
C03337=1181.084,29.994,-46.750,-179.658,5.890,148.949
C03338=1181.079,30.243,-46.765,-179.656,5.891,148.948
C03339=1181.074,30.493,-46.779,-179.653,5.891,148.947
C03340=1181.068,30.742,-46.795,-179.650,5.893,148.947
C03341=1181.064,30.991,-46.810,-179.648,5.893,148.946
C03342=1181.058,31.242,-46.825,-179.645,5.894,148.946
C03343=1181.053,31.491,-46.840,-179.643,5.895,148.945
C03344=1181.049,31.740,-46.855,-179.640,5.895,148.944
C03345=1181.044,31.990,-46.870,-179.638,5.896,148.944
C03346=1181.039,32.240,-46.885,-179.636,5.896,148.943
C03347=1181.034,32.489,-46.901,-179.632,5.898,148.943
C03348=1181.029,32.738,-46.916,-179.630,5.898,148.942
C03349=1181.023,32.988,-46.931,-179.627,5.899,148.942
C03350=1181.019,33.237,-46.946,-179.625,5.900,148.941
C03351=1181.013,33.487,-46.961,-179.622,5.900,148.940
C03352=1181.008,33.736,-46.975,-179.620,5.901,148.940
C03353=1181.004,33.986,-46.991,-179.617,5.902,148.939
C03354=1180.999,34.235,-47.006,-179.615,5.903,148.939
C03355=1180.994,34.485,-47.022,-179.612,5.904,148.938
C03356=1180.989,34.734,-47.037,-179.609,5.904,148.937
C03357=1180.983,34.984,-47.052,-179.607,5.905,148.937
C03358=1180.979,35.233,-47.067,-179.605,5.906,148.936
C03359=1180.973,35.482,-47.082,-179.601,5.907,148.935
C03360=1180.969,35.732,-47.098,-179.599,5.908,148.935
C03361=1180.964,35.982,-47.113,-179.597,5.908,148.934
C03362=1180.958,36.232,-47.128,-179.594,5.909,148.934
C03363=1180.953,36.481,-47.143,-179.592,5.910,148.933
C03364=1180.948,36.730,-47.159,-179.589,5.910,148.933
C03365=1180.943,36.979,-47.174,-179.586,5.912,148.932
C03366=1180.939,37.229,-47.190,-179.584,5.912,148.931
C03367=1180.934,37.478,-47.205,-179.581,5.913,148.931
C03368=1180.929,37.728,-47.220,-179.579,5.914,148.930
C03369=1180.923,37.978,-47.235,-179.576,5.914,148.930
C03370=1180.918,38.227,-47.250,-179.574,5.915,148.929
C03371=1180.913,38.477,-47.266,-179.571,5.916,148.929
C03372=1180.908,38.726,-47.282,-179.568,5.917,148.928
C03373=1180.903,38.976,-47.297,-179.566,5.918,148.927
C03374=1180.898,39.225,-47.312,-179.563,5.918,148.927
C03375=1180.893,39.474,-47.327,-179.561,5.919,148.926
C03376=1180.889,39.724,-47.343,-179.558,5.920,148.926
C03377=1180.883,39.974,-47.359,-179.555,5.921,148.925
C03378=1180.879,40.223,-47.374,-179.553,5.921,148.924
C03379=1180.873,40.472,-47.389,-179.551,5.922,148.924
C03380=1180.868,40.721,-47.405,-179.548,5.923,148.923
C03381=1180.864,40.971,-47.420,-179.545,5.924,148.923
C03382=1180.858,41.221,-47.436,-179.543,5.925,148.922
C03383=1180.853,41.470,-47.452,-179.540,5.925,148.921
C03384=1180.848,41.719,-47.467,-179.538,5.926,148.921
C03385=1180.843,41.969,-47.483,-179.535,5.927,148.920
C03386=1180.838,42.219,-47.498,-179.532,5.928,148.920
C03387=1180.833,42.468,-47.514,-179.530,5.929,148.919
C03388=1180.829,42.718,-47.529,-179.527,5.930,148.918
C03389=1180.823,42.967,-47.545,-179.525,5.930,148.918
C03390=1180.818,43.217,-47.560,-179.522,5.931,148.917
C03391=1180.812,43.466,-47.576,-179.519,5.932,148.917
C03392=1180.808,43.716,-47.591,-179.517,5.933,148.916
C03393=1180.803,43.965,-47.608,-179.514,5.934,148.916
C03394=1180.798,44.214,-47.623,-179.512,5.934,148.915
C03395=1180.793,44.464,-47.639,-179.509,5.936,148.914
C03396=1180.789,44.713,-47.654,-179.506,5.936,148.914
C03397=1180.783,44.963,-47.670,-179.504,5.937,148.913
C03398=1180.778,45.212,-47.685,-179.502,5.938,148.913
C03399=1180.773,45.462,-47.701,-179.499,5.938,148.912
C03400=1180.769,45.711,-47.717,-179.496,5.940,148.912
C03401=1180.763,45.960,-47.732,-179.493,5.940,148.911
C03402=1180.758,46.210,-47.748,-179.491,5.941,148.910
C03403=1180.753,46.460,-47.764,-179.489,5.942,148.910
C03404=1180.748,46.709,-47.780,-179.485,5.943,148.909
C03405=1180.743,46.958,-47.796,-179.483,5.944,148.909
C03406=1180.739,47.207,-47.811,-179.481,5.944,148.908
C03407=1180.733,47.457,-47.827,-179.479,5.945,148.908
C03408=1180.728,47.707,-47.843,-179.475,5.947,148.907
C03409=1180.723,47.956,-47.859,-179.473,5.947,148.906
C03410=1180.719,48.206,-47.875,-179.471,5.948,148.906
C03411=1180.713,48.455,-47.891,-179.468,5.949,148.905
C03412=1180.708,48.704,-47.906,-179.466,5.949,148.905
C03413=1180.704,48.954,-47.922,-179.462,5.951,148.904
C03414=1180.699,49.203,-47.938,-179.460,5.951,148.903
C03415=1180.693,49.453,-47.953,-179.458,5.952,148.903
C03416=1180.689,49.702,-47.970,-179.455,5.953,148.902
C03417=1180.683,49.952,-47.986,-179.452,5.954,148.902
C03418=1180.679,50.202,-48.002,-179.450,5.955,148.901
C03419=1180.674,50.450,-48.018,-179.447,5.955,148.900
C03420=1180.668,50.700,-48.034,-179.444,5.957,148.900
C03421=1180.663,50.950,-48.050,-179.442,5.958,148.899
C03422=1180.659,51.198,-48.065,-179.440,5.958,148.899
C03423=1180.654,51.449,-48.081,-179.437,5.959,148.898
C03424=1180.649,51.698,-48.097,-179.434,5.961,148.898
C03425=1180.644,51.947,-48.113,-179.432,5.961,148.897
C03426=1180.639,52.197,-48.129,-179.429,5.962,148.896
C03427=1180.634,52.446,-48.145,-179.427,5.963,148.896
C03428=1180.629,52.696,-48.161,-179.424,5.964,148.895
C03429=1180.624,52.944,-48.178,-179.421,5.965,148.895
C03430=1180.619,53.195,-48.194,-179.419,5.965,148.894
C03431=1180.614,53.444,-48.209,-179.416,5.966,148.894
C03432=1180.609,53.693,-48.226,-179.413,5.968,148.893
C03433=1180.604,53.943,-48.241,-179.411,5.968,148.892
C03434=1180.599,54.211,-48.259,-179.408,5.969,148.892
C03435=1180.594,54.480,-48.277,-179.405,5.970,148.891
C03436=1180.588,54.748,-48.294,-179.403,5.971,148.891
C03437=1180.583,55.017,-48.311,-179.399,5.972,148.890
C03438=1180.578,55.266,-48.327,-179.397,5.973,148.890
C03439=1180.572,55.516,-48.343,-179.395,5.973,148.889
C03440=1180.568,55.766,-48.360,-179.391,5.975,148.888
C03441=1180.562,56.014,-48.376,-179.389,5.976,148.888
C03442=1180.558,56.264,-48.392,-179.387,5.976,148.887
C03443=1180.553,56.513,-48.409,-179.384,5.978,148.887
C03444=1180.548,56.763,-48.425,-179.381,5.978,148.886
C03445=1180.543,57.012,-48.441,-179.379,5.979,148.886
C03446=1180.538,57.262,-48.457,-179.377,5.980,148.885
C03447=1180.533,57.511,-48.473,-179.373,5.981,148.884
C03448=1180.528,57.760,-48.490,-179.371,5.982,148.884
C03449=1180.523,58.010,-48.505,-179.369,5.983,148.883
C03450=1180.519,58.259,-48.522,-179.366,5.984,148.883
C03451=1180.513,58.508,-48.539,-179.363,5.985,148.882
C03452=1180.508,58.759,-48.555,-179.361,5.986,148.882
C03453=1180.503,59.007,-48.571,-179.358,5.987,148.881
C03454=1180.498,59.257,-48.587,-179.355,5.987,148.880
C03455=1180.493,59.506,-48.603,-179.353,5.988,148.880
C03456=1180.488,59.756,-48.620,-179.350,5.989,148.879
C03457=1180.483,60.004,-48.636,-179.348,5.991,148.879
C03458=1180.478,60.255,-48.653,-179.345,5.991,148.878
C03459=1180.473,60.504,-48.670,-179.343,5.992,148.878
C03460=1180.468,60.753,-48.686,-179.340,5.993,148.877
C03461=1180.464,61.003,-48.702,-179.337,5.994,148.877
C03462=1180.458,61.252,-48.718,-179.335,5.995,148.876
C03463=1180.453,61.502,-48.735,-179.332,5.996,148.875
C03464=1180.449,61.751,-48.752,-179.329,5.997,148.875
C03465=1180.443,62.001,-48.768,-179.327,5.997,148.874
C03466=1180.439,62.250,-48.784,-179.324,5.999,148.874
C03467=1180.434,62.499,-48.801,-179.321,6.000,148.873
C03468=1180.429,62.749,-48.818,-179.319,6.001,148.873
C03469=1180.424,62.998,-48.835,-179.316,6.002,148.872
C03470=1180.419,63.248,-48.850,-179.314,6.003,148.871
C03471=1180.414,63.497,-48.867,-179.311,6.003,148.871
C03472=1180.408,63.746,-48.884,-179.308,6.005,148.870
C03473=1180.404,63.996,-48.900,-179.306,6.006,148.870
C03474=1180.399,64.245,-48.917,-179.303,6.006,148.869
C03475=1180.394,64.494,-48.933,-179.301,6.008,148.869
C03476=1180.389,64.744,-48.950,-179.298,6.008,148.868
C03477=1180.384,64.994,-48.967,-179.296,6.009,148.868
C03478=1180.379,65.243,-48.983,-179.293,6.010,148.867
C03479=1180.375,65.492,-49.000,-179.290,6.011,148.866
C03480=1180.370,65.742,-49.017,-179.288,6.012,148.866
C03481=1180.365,65.991,-49.033,-179.285,6.014,148.865
C03482=1180.360,66.240,-49.050,-179.282,6.014,148.865
C03483=1180.355,66.490,-49.067,-179.280,6.015,148.864
C03484=1180.350,66.739,-49.083,-179.277,6.016,148.864
C03485=1180.345,66.988,-49.100,-179.274,6.017,148.863
C03486=1180.340,67.238,-49.117,-179.272,6.018,148.863
C03487=1180.335,67.487,-49.134,-179.269,6.019,148.862
C03488=1180.330,67.736,-49.150,-179.267,6.020,148.861
C03489=1180.325,67.986,-49.168,-179.264,6.021,148.861
C03490=1180.320,68.235,-49.184,-179.262,6.022,148.860
C03491=1180.315,68.485,-49.201,-179.259,6.023,148.860
C03492=1180.310,68.734,-49.218,-179.256,6.024,148.859
C03493=1180.305,68.983,-49.234,-179.254,6.025,148.859
C03494=1180.300,69.233,-49.251,-179.251,6.026,148.858
C03495=1180.296,69.482,-49.268,-179.248,6.027,148.857
C03496=1180.291,69.732,-49.285,-179.246,6.028,148.857
C03497=1180.285,69.981,-49.302,-179.243,6.029,148.856
C03498=1180.281,70.230,-49.318,-179.241,6.030,148.856
C03499=1180.276,70.480,-49.336,-179.238,6.031,148.855
C03500=1180.271,70.730,-49.352,-179.235,6.033,148.855
C03501=1180.265,70.979,-49.369,-179.233,6.033,148.854
C03502=1180.261,71.228,-49.386,-179.230,6.034,148.854
C03503=1180.256,71.478,-49.403,-179.227,6.035,148.853
C03504=1180.252,71.727,-49.420,-179.225,6.036,148.852
C03505=1180.246,71.976,-49.437,-179.222,6.038,148.852
C03506=1180.241,72.225,-49.454,-179.219,6.038,148.851
C03507=1180.237,72.475,-49.471,-179.217,6.039,148.851
C03508=1180.232,72.725,-49.488,-179.214,6.040,148.850
C03509=1180.226,72.974,-49.504,-179.212,6.041,148.850
C03510=1180.222,73.223,-49.522,-179.209,6.043,148.849
C03511=1180.217,73.472,-49.539,-179.207,6.043,148.849
C03512=1180.212,73.722,-49.556,-179.204,6.044,148.848
C03513=1180.207,73.971,-49.573,-179.201,6.046,148.848
C03514=1180.202,74.221,-49.590,-179.199,6.046,148.847
C03515=1180.197,74.469,-49.607,-179.196,6.048,148.847
C03516=1180.192,74.719,-49.624,-179.193,6.048,148.846
C03517=1180.187,74.969,-49.642,-179.191,6.049,148.846
C03518=1180.182,75.218,-49.658,-179.188,6.051,148.845
C03519=1180.177,75.467,-49.676,-179.186,6.052,148.844
C03520=1180.172,75.716,-49.693,-179.183,6.053,148.844
C03521=1180.167,75.966,-49.710,-179.180,6.054,148.843
C03522=1180.163,76.215,-49.727,-179.178,6.054,148.843
C03523=1180.158,76.465,-49.745,-179.175,6.056,148.842
C03524=1180.153,76.715,-49.762,-179.172,6.057,148.842
C03525=1180.148,76.963,-49.779,-179.170,6.058,148.841
C03526=1180.143,77.213,-49.796,-179.167,6.059,148.841
C03527=1180.138,77.462,-49.813,-179.165,6.060,148.840
C03528=1180.133,77.711,-49.831,-179.162,6.061,148.839
C03529=1180.128,77.961,-49.848,-179.160,6.062,148.839
C03530=1180.124,78.211,-49.865,-179.156,6.063,148.838
C03531=1180.119,78.460,-49.883,-179.154,6.064,148.838
C03532=1180.113,78.709,-49.900,-179.151,6.066,148.837
C03533=1180.108,78.958,-49.916,-179.149,6.066,148.837
C03534=1180.103,79.208,-49.934,-179.146,6.067,148.836
C03535=1180.098,79.457,-49.951,-179.144,6.069,148.836
C03536=1180.094,79.706,-49.969,-179.141,6.069,148.835
C03537=1180.089,79.956,-49.986,-179.138,6.071,148.835
C03538=1180.084,80.224,-50.006,-179.136,6.071,148.834
C03539=1180.078,80.492,-50.023,-179.133,6.073,148.834
C03540=1180.073,80.761,-50.042,-179.130,6.075,148.833
C03541=1180.068,81.029,-50.061,-179.127,6.075,148.832
C03542=1180.063,81.279,-50.079,-179.124,6.077,148.832
C03543=1180.059,81.528,-50.096,-179.122,6.077,148.831
C03544=1180.053,81.778,-50.113,-179.119,6.079,148.831
C03545=1180.049,82.027,-50.131,-179.116,6.080,148.830
C03546=1180.043,82.276,-50.148,-179.114,6.080,148.830
C03547=1180.039,82.525,-50.166,-179.111,6.082,148.829
C03548=1180.033,82.775,-50.183,-179.109,6.083,148.829
C03549=1180.028,83.024,-50.201,-179.106,6.084,148.828
C03550=1180.023,83.274,-50.218,-179.103,6.085,148.828
C03551=1180.019,83.522,-50.235,-179.101,6.087,148.827
C03552=1180.014,83.772,-50.253,-179.098,6.087,148.827
C03553=1180.009,84.021,-50.271,-179.095,6.089,148.826
C03554=1180.004,84.271,-50.289,-179.093,6.089,148.825
C03555=1179.999,84.520,-50.306,-179.090,6.091,148.825
C03556=1179.995,84.769,-50.323,-179.087,6.092,148.824
C03557=1179.990,85.018,-50.341,-179.085,6.093,148.824
C03558=1179.984,85.268,-50.359,-179.082,6.094,148.823
C03559=1179.980,85.517,-50.377,-179.079,6.096,148.823
C03560=1179.975,85.767,-50.395,-179.077,6.096,148.822
C03561=1179.969,86.016,-50.412,-179.075,6.097,148.822
C03562=1179.965,86.265,-50.429,-179.072,6.099,148.821
C03563=1179.960,86.514,-50.447,-179.069,6.099,148.821
C03564=1179.955,86.764,-50.464,-179.067,6.101,148.820
C03565=1179.950,87.013,-50.482,-179.064,6.102,148.820
C03566=1179.945,87.263,-50.500,-179.061,6.103,148.819
C03567=1179.940,87.512,-50.518,-179.059,6.104,148.819
C03568=1179.935,87.762,-50.536,-179.056,6.106,148.818
C03569=1179.931,88.010,-50.553,-179.053,6.106,148.818
C03570=1179.926,88.260,-50.571,-179.050,6.108,148.817
C03571=1179.921,88.509,-50.589,-179.048,6.108,148.816
C03572=1179.916,88.759,-50.606,-179.045,6.110,148.816
C03573=1179.911,89.008,-50.624,-179.043,6.111,148.816
C03574=1179.906,89.257,-50.642,-179.040,6.112,148.815
C03575=1179.902,89.507,-50.661,-179.038,6.113,148.815
C03576=1179.897,89.756,-50.679,-179.034,6.115,148.814
C03577=1179.892,90.006,-50.696,-179.032,6.116,148.813
C03578=1179.887,90.255,-50.714,-179.029,6.117,148.813
C03579=1179.882,90.504,-50.732,-179.027,6.118,148.812
C03580=1179.877,90.753,-50.750,-179.024,6.120,148.812
C03581=1179.872,91.002,-50.768,-179.022,6.120,148.811
C03582=1179.867,91.252,-50.786,-179.019,6.122,148.811
C03583=1179.862,91.501,-50.804,-179.016,6.122,148.810
C03584=1179.857,91.750,-50.822,-179.014,6.124,148.810
C03585=1179.852,92.000,-50.839,-179.011,6.125,148.809
C03586=1179.848,92.250,-50.857,-179.008,6.126,148.809
C03587=1179.843,92.499,-50.875,-179.006,6.127,148.808
C03588=1179.838,92.748,-50.893,-179.003,6.129,148.808
C03589=1179.833,92.997,-50.911,-179.001,6.129,148.807
C03590=1179.828,93.246,-50.929,-178.998,6.131,148.807
C03591=1179.823,93.495,-50.947,-178.995,6.132,148.806
C03592=1179.818,93.745,-50.965,-178.992,6.133,148.806
C03593=1179.813,93.994,-50.983,-178.990,6.134,148.805
C03594=1179.809,94.244,-51.001,-178.987,6.136,148.805
C03595=1179.804,94.493,-51.019,-178.984,6.137,148.804
C03596=1179.799,94.742,-51.037,-178.982,6.138,148.804
C03597=1179.794,94.991,-51.055,-178.979,6.139,148.803
C03598=1179.789,95.240,-51.073,-178.977,6.140,148.803
C03599=1179.784,95.490,-51.091,-178.974,6.142,148.802
C03600=1179.779,95.740,-51.110,-178.971,6.143,148.802
C03601=1179.775,95.989,-51.128,-178.969,6.144,148.801
C03602=1179.770,96.238,-51.146,-178.966,6.145,148.801
C03603=1179.765,96.487,-51.165,-178.963,6.147,148.800
C03604=1179.760,96.736,-51.183,-178.961,6.147,148.800
C03605=1179.756,96.986,-51.201,-178.958,6.149,148.799
C03606=1179.751,97.235,-51.219,-178.956,6.150,148.799
C03607=1179.746,97.484,-51.237,-178.953,6.151,148.798
C03608=1179.740,97.734,-51.256,-178.950,6.153,148.798
C03609=1179.735,97.983,-51.274,-178.948,6.154,148.797
C03610=1179.731,98.233,-51.292,-178.945,6.155,148.797
C03611=1179.726,98.481,-51.311,-178.942,6.156,148.796
C03612=1179.722,98.730,-51.329,-178.939,6.157,148.795
C03613=1179.717,98.980,-51.347,-178.937,6.158,148.795
C03614=1179.711,99.229,-51.365,-178.934,6.160,148.795
C03615=1179.707,99.479,-51.384,-178.932,6.161,148.794
C03616=1179.702,99.727,-51.402,-178.929,6.162,148.794
C03617=1179.697,99.977,-51.420,-178.926,6.164,148.793
C03618=1179.692,100.226,-51.439,-178.924,6.165,148.793
C03619=1179.687,100.476,-51.457,-178.921,6.166,148.792
C03620=1179.683,100.725,-51.476,-178.918,6.167,148.791
C03621=1179.678,100.974,-51.494,-178.916,6.169,148.791
C03622=1179.673,101.224,-51.512,-178.913,6.169,148.790
C03623=1179.668,101.473,-51.531,-178.910,6.171,148.790
C03624=1179.663,101.722,-51.550,-178.908,6.173,148.790
C03625=1179.658,101.971,-51.568,-178.905,6.173,148.789
C03626=1179.653,102.221,-51.587,-178.902,6.175,148.789
C03627=1179.649,102.470,-51.605,-178.900,6.176,148.788
C03628=1179.644,102.719,-51.623,-178.897,6.177,148.787
C03629=1179.639,102.969,-51.642,-178.895,6.178,148.787
C03630=1179.634,103.217,-51.661,-178.892,6.179,148.786
C03631=1179.629,103.467,-51.679,-178.889,6.181,148.786
C03632=1179.624,103.716,-51.697,-178.887,6.182,148.786
C03633=1179.619,103.965,-51.716,-178.884,6.183,148.785
C03634=1179.615,104.215,-51.734,-178.881,6.184,148.785
C03635=1179.610,104.463,-51.753,-178.879,6.186,148.784
C03636=1179.605,104.713,-51.772,-178.876,6.187,148.784
C03637=1179.600,104.963,-51.790,-178.873,6.188,148.783
C03638=1179.595,105.211,-51.809,-178.871,6.190,148.783
C03639=1179.590,105.461,-51.828,-178.868,6.191,148.782
C03640=1179.586,105.710,-51.846,-178.865,6.192,148.782
C03641=1179.580,105.959,-51.865,-178.862,6.194,148.781
C03642=1179.576,106.228,-51.885,-178.860,6.195,148.781
C03643=1179.570,106.496,-51.905,-178.857,6.196,148.780
C03644=1179.565,106.764,-51.925,-178.854,6.198,148.780
C03645=1179.560,107.033,-51.946,-178.851,6.199,148.779
C03646=1179.555,107.282,-51.964,-178.849,6.200,148.779
C03647=1179.550,107.531,-51.983,-178.846,6.202,148.778
C03648=1179.545,107.781,-52.002,-178.843,6.203,148.777
C03649=1179.540,108.030,-52.021,-178.841,6.204,148.777
C03650=1179.536,108.280,-52.039,-178.838,6.206,148.777
C03651=1179.530,108.529,-52.058,-178.835,6.207,148.776
C03652=1179.526,108.777,-52.077,-178.833,6.208,148.776
C03653=1179.522,109.027,-52.096,-178.830,6.210,148.775
C03654=1179.516,109.276,-52.115,-178.827,6.210,148.775
C03655=1179.512,109.526,-52.133,-178.825,6.212,148.774
C03656=1179.507,109.775,-52.152,-178.822,6.214,148.774
C03657=1179.503,110.024,-52.171,-178.819,6.214,148.773
C03658=1179.497,110.273,-52.190,-178.817,6.216,148.773
